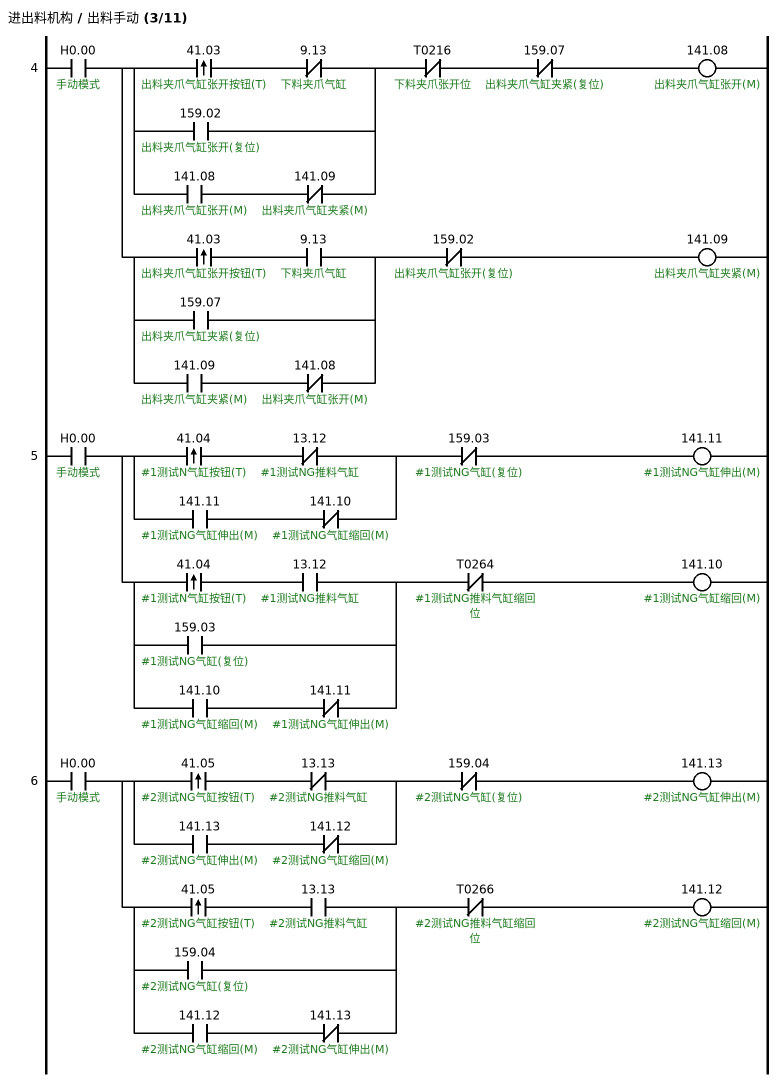
; [picture p96: 进出料机构 / 出料手动, rungs 4-6]
; rung 4
LD H0.00  ; 手动模式
OUT TR0
@LD 41.03  ; 出料夹爪气缸张开按钮(T)
ANDNOT 9.13  ; 下料夹爪气缸
OR 159.02  ; 出料夹爪气缸张开(复位)
LD 141.08  ; 出料夹爪气缸张开(M)
ANDNOT 141.09  ; 出料夹爪气缸夹紧(M)
ORLD
ANDLD
ANDNOT T0216  ; 下料夹爪张开位
ANDNOT 159.07  ; 出料夹爪气缸夹紧(复位)
OUT 141.08  ; 出料夹爪气缸张开(M)
LD TR0
@LD 41.03  ; 出料夹爪气缸张开按钮(T)
AND 9.13  ; 下料夹爪气缸
OR 159.07  ; 出料夹爪气缸夹紧(复位)
LD 141.09  ; 出料夹爪气缸夹紧(M)
ANDNOT 141.08  ; 出料夹爪气缸张开(M)
ORLD
ANDLD
ANDNOT 159.02  ; 出料夹爪气缸张开(复位)
OUT 141.09  ; 出料夹爪气缸夹紧(M)
; rung 5
LD H0.00  ; 手动模式
OUT TR0
@LD 41.04  ; #1测试N气缸按钮(T)
ANDNOT 13.12  ; #1测试NG推料气缸
LD 141.11  ; #1测试NG气缸伸出(M)
ANDNOT 141.10  ; #1测试NG气缸缩回(M)
ORLD
ANDLD
ANDNOT 159.03  ; #1测试NG气缸(复位)
OUT 141.11  ; #1测试NG气缸伸出(M)
LD TR0
@LD 41.04  ; #1测试N气缸按钮(T)
AND 13.12  ; #1测试NG推料气缸
OR 159.03  ; #1测试NG气缸(复位)
LD 141.10  ; #1测试NG气缸缩回(M)
ANDNOT 141.11  ; #1测试NG气缸伸出(M)
ORLD
ANDLD
ANDNOT T0264  ; #1测试NG推料气缸缩回位
OUT 141.10  ; #1测试NG气缸缩回(M)
; rung 6
LD H0.00  ; 手动模式
OUT TR0
@LD 41.05  ; #2测试NG气缸按钮(T)
ANDNOT 13.13  ; #2测试NG推料气缸
LD 141.13  ; #2测试NG气缸伸出(M)
ANDNOT 141.12  ; #2测试NG气缸缩回(M)
ORLD
ANDLD
ANDNOT 159.04  ; #2测试NG气缸(复位)
OUT 141.13  ; #2测试NG气缸伸出(M)
LD TR0
@LD 41.05  ; #2测试NG气缸按钮(T)
AND 13.13  ; #2测试NG推料气缸
OR 159.04  ; #2测试NG气缸(复位)
LD 141.12  ; #2测试NG气缸缩回(M)
ANDNOT 141.13  ; #2测试NG气缸伸出(M)
ORLD
ANDLD
ANDNOT T0266  ; #2测试NG推料气缸缩回位
OUT 141.12  ; #2测试NG气缸缩回(M)

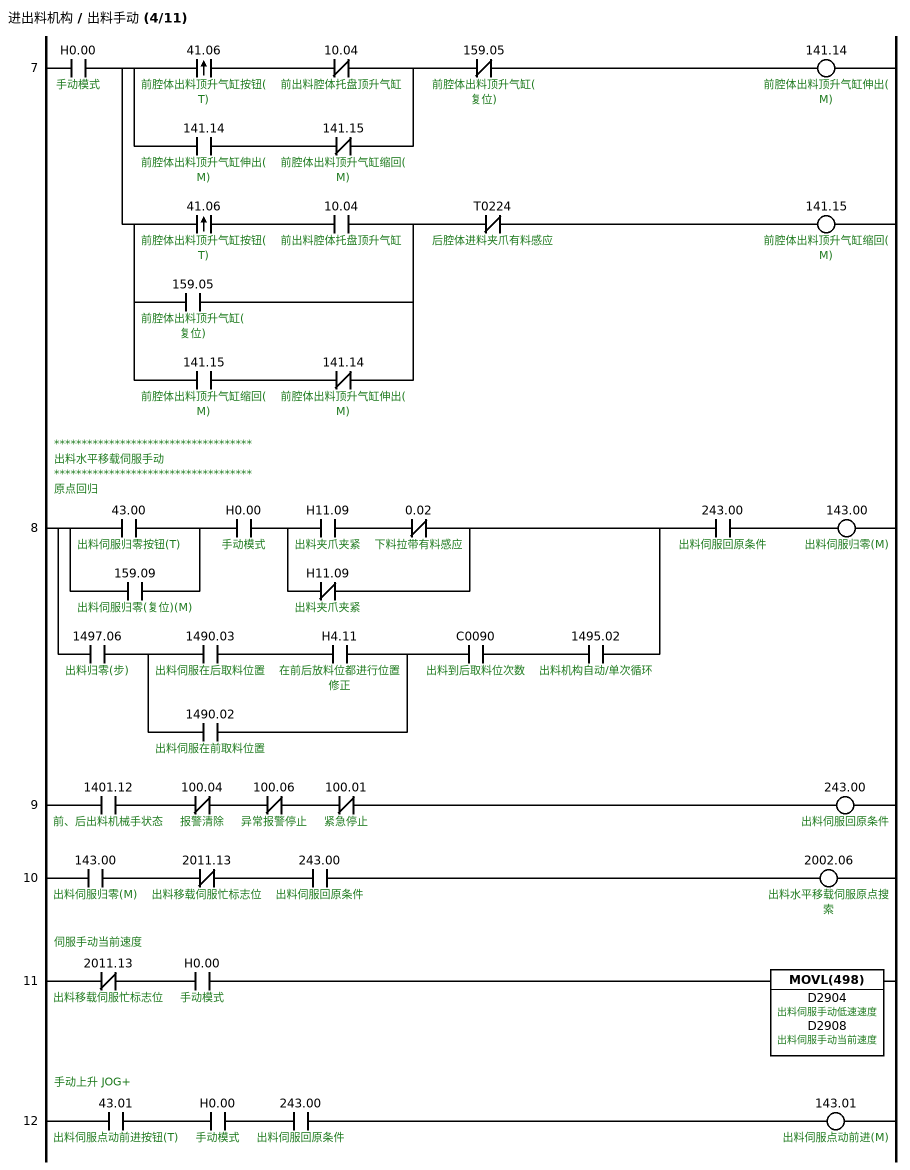
; rung 7
LD H0.00  ; 手动模式
OUT TR0
@LD 41.06  ; 前腔体出料顶升气缸按钮(T)
ANDNOT 10.04  ; 前出料腔体托盘顶升气缸
LD 141.14  ; 前腔体出料顶升气缸伸出(M)
ANDNOT 141.15  ; 前腔体出料顶升气缸缩回(M)
ORLD
ANDLD
ANDNOT 159.05  ; 前腔体出料顶升气缸(复位)
OUT 141.14  ; 前腔体出料顶升气缸伸出(M)
LD TR0
@LD 41.06  ; 前腔体出料顶升气缸按钮(T)
AND 10.04  ; 前出料腔体托盘顶升气缸
OR 159.05  ; 前腔体出料顶升气缸(复位)
LD 141.15  ; 前腔体出料顶升气缸缩回(M)
ANDNOT 141.14  ; 前腔体出料顶升气缸伸出(M)
ORLD
ANDLD
ANDNOT T0224  ; 后腔体进料夹爪有料感应
OUT 141.15  ; 前腔体出料顶升气缸缩回(M)
; rung 8: ************************************ / 出料水平移载伺服手动 / ************************************ / 原点回归
LD 43.00  ; 出料伺服归零按钮(T)
OR 159.09  ; 出料伺服归零(复位)(M)
AND H0.00  ; 手动模式
LD H11.09  ; 出料夹爪夹紧
ANDNOT 0.02  ; 下料拉带有料感应
ORNOT H11.09  ; 出料夹爪夹紧
ANDLD
LD 1497.06  ; 出料归零(步)
LD 1490.03  ; 出料伺服在后取料位置
AND H4.11  ; 在前后放料位都进行位置修正
OR 1490.02  ; 出料伺服在前取料位置
ANDLD
AND C0090  ; 出料到后取料位次数
AND 1495.02  ; 出料机构自动/单次循环
ORLD
AND 243.00  ; 出料伺服回原条件
OUT 143.00  ; 出料伺服归零(M)
; rung 9
LD 1401.12  ; 前、后出料机械手状态
ANDNOT 100.04  ; 报警清除
ANDNOT 100.06  ; 异常报警停止
ANDNOT 100.01  ; 紧急停止
OUT 243.00  ; 出料伺服回原条件
; rung 10
LD 143.00  ; 出料伺服归零(M)
ANDNOT 2011.13  ; 出料移载伺服忙标志位
AND 243.00  ; 出料伺服回原条件
OUT 2002.06  ; 出料水平移载伺服原点搜索
; rung 11: 伺服手动当前速度
LDNOT 2011.13  ; 出料移载伺服忙标志位
AND H0.00  ; 手动模式
MOVL(498) D2904 D2908  ; 出料伺服手动低速速度, 出料伺服手动当前速度
; rung 12: 手动上升 JOG+
LD 43.01  ; 出料伺服点动前进按钮(T)
AND H0.00  ; 手动模式
AND 243.00  ; 出料伺服回原条件
OUT 143.01  ; 出料伺服点动前进(M)

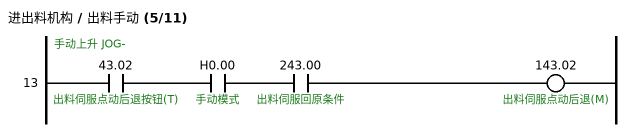
; rung 13: 手动上升 JOG-
LD 43.02  ; 出料伺服点动后退按钮(T)
AND H0.00  ; 手动模式
AND 243.00  ; 出料伺服回原条件
OUT 143.02  ; 出料伺服点动后退(M)

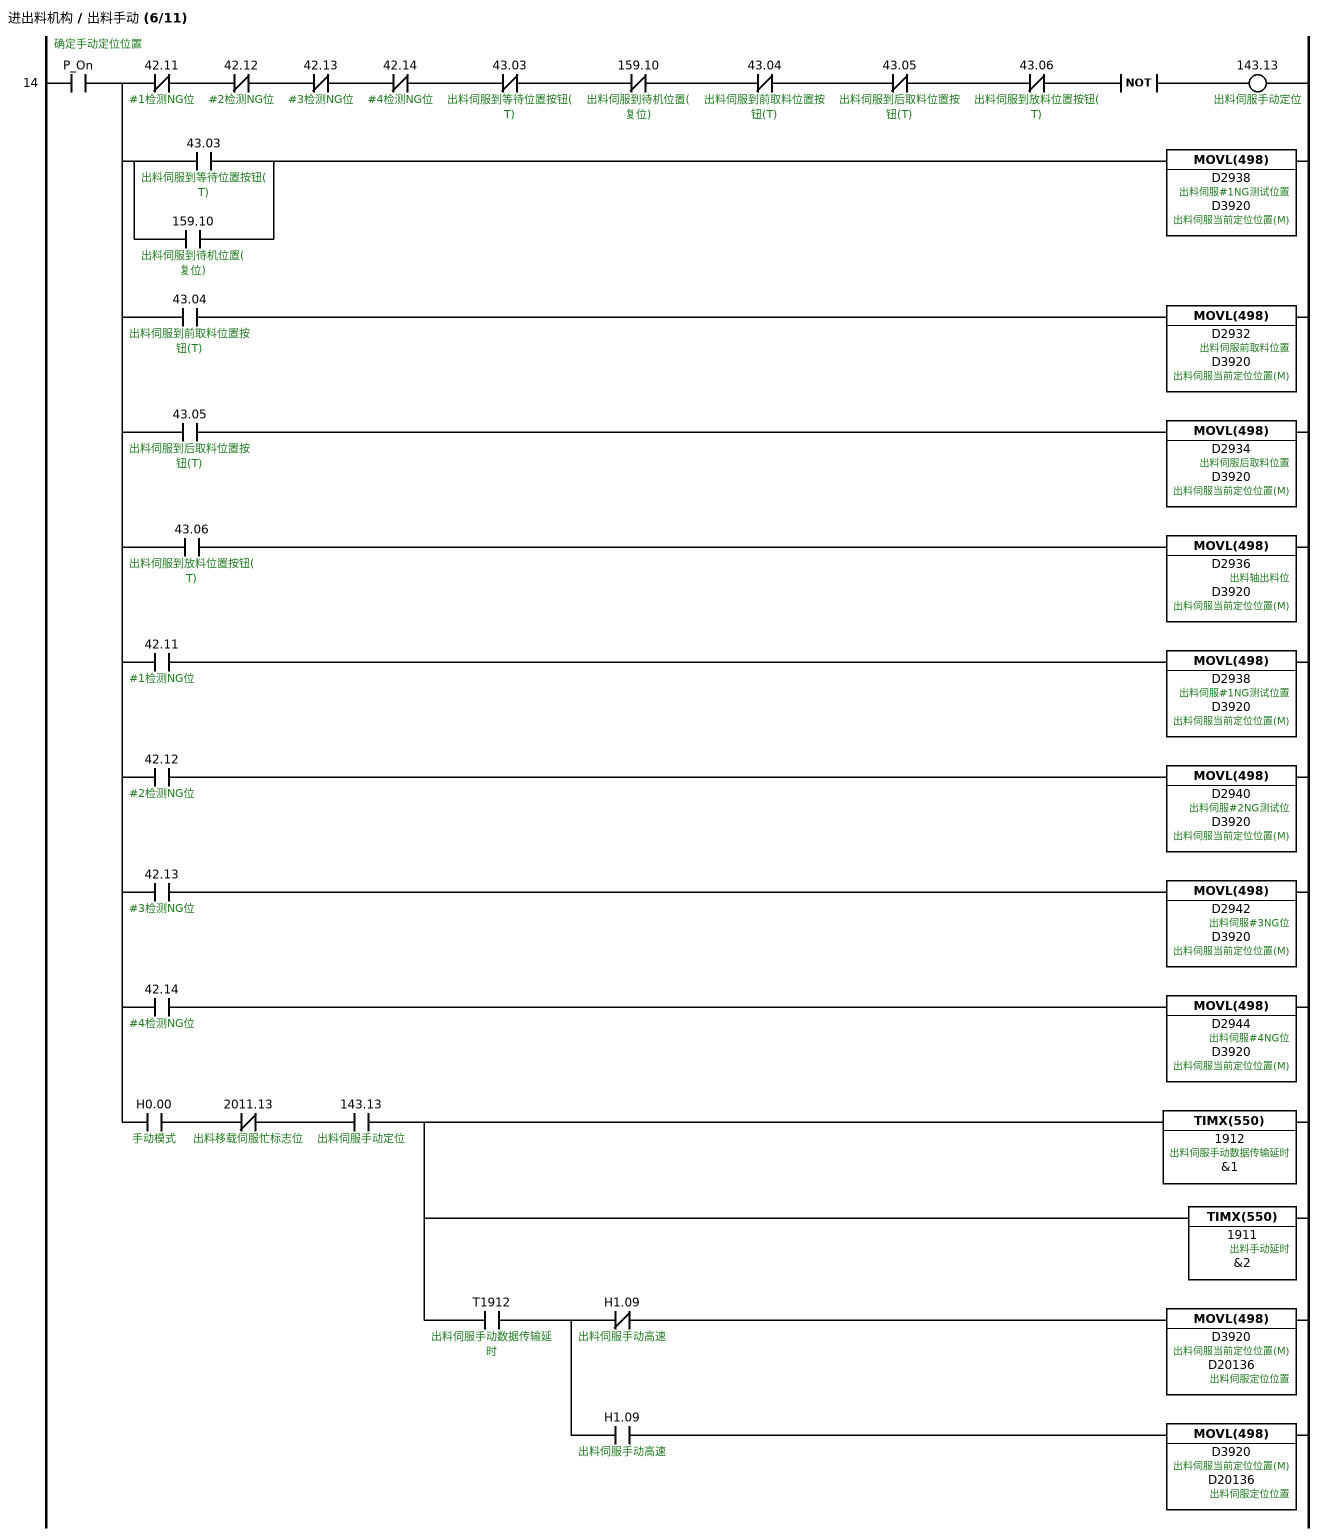
; rung 14: 确定手动定位位置
LD P_On
OUT TR0
ANDNOT 42.11  ; #1检测NG位
ANDNOT 42.12  ; #2检测NG位
ANDNOT 42.13  ; #3检测NG位
ANDNOT 42.14  ; #4检测NG位
ANDNOT 43.03  ; 出料伺服到等待位置按钮(T)
ANDNOT 159.10  ; 出料伺服到待机位置(复位)
ANDNOT 43.04  ; 出料伺服到前取料位置按钮(T)
ANDNOT 43.05  ; 出料伺服到后取料位置按钮(T)
ANDNOT 43.06  ; 出料伺服到放料位置按钮(T)
NOT(520)
OUT 143.13  ; 出料伺服手动定位
LD TR0
LD 43.03  ; 出料伺服到等待位置按钮(T)
OR 159.10  ; 出料伺服到待机位置(复位)
ANDLD
MOVL(498) D2938 D3920  ; 出料伺服#1NG测试位置, 出料伺服当前定位位置(M)
LD TR0
AND 43.04  ; 出料伺服到前取料位置按钮(T)
MOVL(498) D2932 D3920  ; 出料伺服前取料位置, 出料伺服当前定位位置(M)
LD TR0
AND 43.05  ; 出料伺服到后取料位置按钮(T)
MOVL(498) D2934 D3920  ; 出料伺服后取料位置, 出料伺服当前定位位置(M)
LD TR0
AND 43.06  ; 出料伺服到放料位置按钮(T)
MOVL(498) D2936 D3920  ; 出料轴出料位, 出料伺服当前定位位置(M)
LD TR0
AND 42.11  ; #1检测NG位
MOVL(498) D2938 D3920  ; 出料伺服#1NG测试位置, 出料伺服当前定位位置(M)
LD TR0
AND 42.12  ; #2检测NG位
MOVL(498) D2940 D3920  ; 出料伺服#2NG测试位, 出料伺服当前定位位置(M)
LD TR0
AND 42.13  ; #3检测NG位
MOVL(498) D2942 D3920  ; 出料伺服#3NG位, 出料伺服当前定位位置(M)
LD TR0
AND 42.14  ; #4检测NG位
MOVL(498) D2944 D3920  ; 出料伺服#4NG位, 出料伺服当前定位位置(M)
LD TR0
AND H0.00  ; 手动模式
ANDNOT 2011.13  ; 出料移载伺服忙标志位
AND 143.13  ; 出料伺服手动定位
TIMX(550) 1912 &1  ; 出料伺服手动数据传输延时
TIMX(550) 1911 &2  ; 出料手动延时
AND T1912  ; 出料伺服手动数据传输延时
OUT TR0
ANDNOT H1.09  ; 出料伺服手动高速
MOVL(498) D3920 D20136  ; 出料伺服当前定位位置(M), 出料伺服定位位置
LD TR0
AND H1.09  ; 出料伺服手动高速
MOVL(498) D3920 D20136  ; 出料伺服当前定位位置(M), 出料伺服定位位置

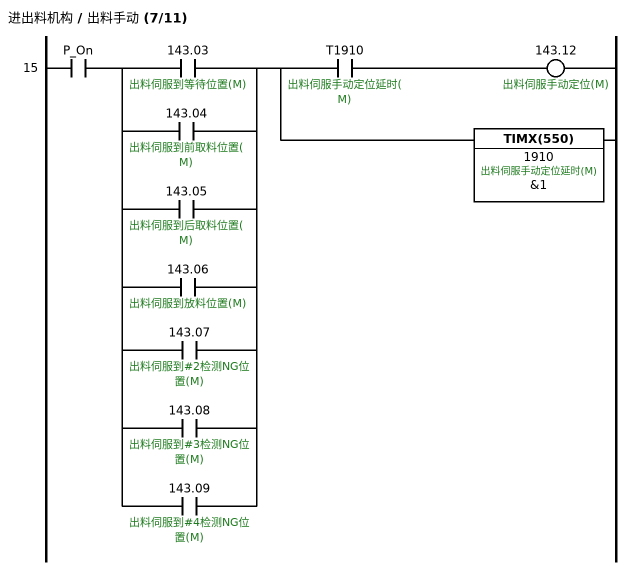
; rung 15
LD P_On
LD 143.03  ; 出料伺服到等待位置(M)
OR 143.04  ; 出料伺服到前取料位置(M)
OR 143.05  ; 出料伺服到后取料位置(M)
OR 143.06  ; 出料伺服到放料位置(M)
OR 143.07  ; 出料伺服到#2检测NG位置(M)
OR 143.08  ; 出料伺服到#3检测NG位置(M)
OR 143.09  ; 出料伺服到#4检测NG位置(M)
ANDLD
OUT TR0
AND T1910  ; 出料伺服手动定位延时(M)
OUT 143.12  ; 出料伺服手动定位(M)
LD TR0
TIMX(550) 1910 &1  ; 出料伺服手动定位延时(M)

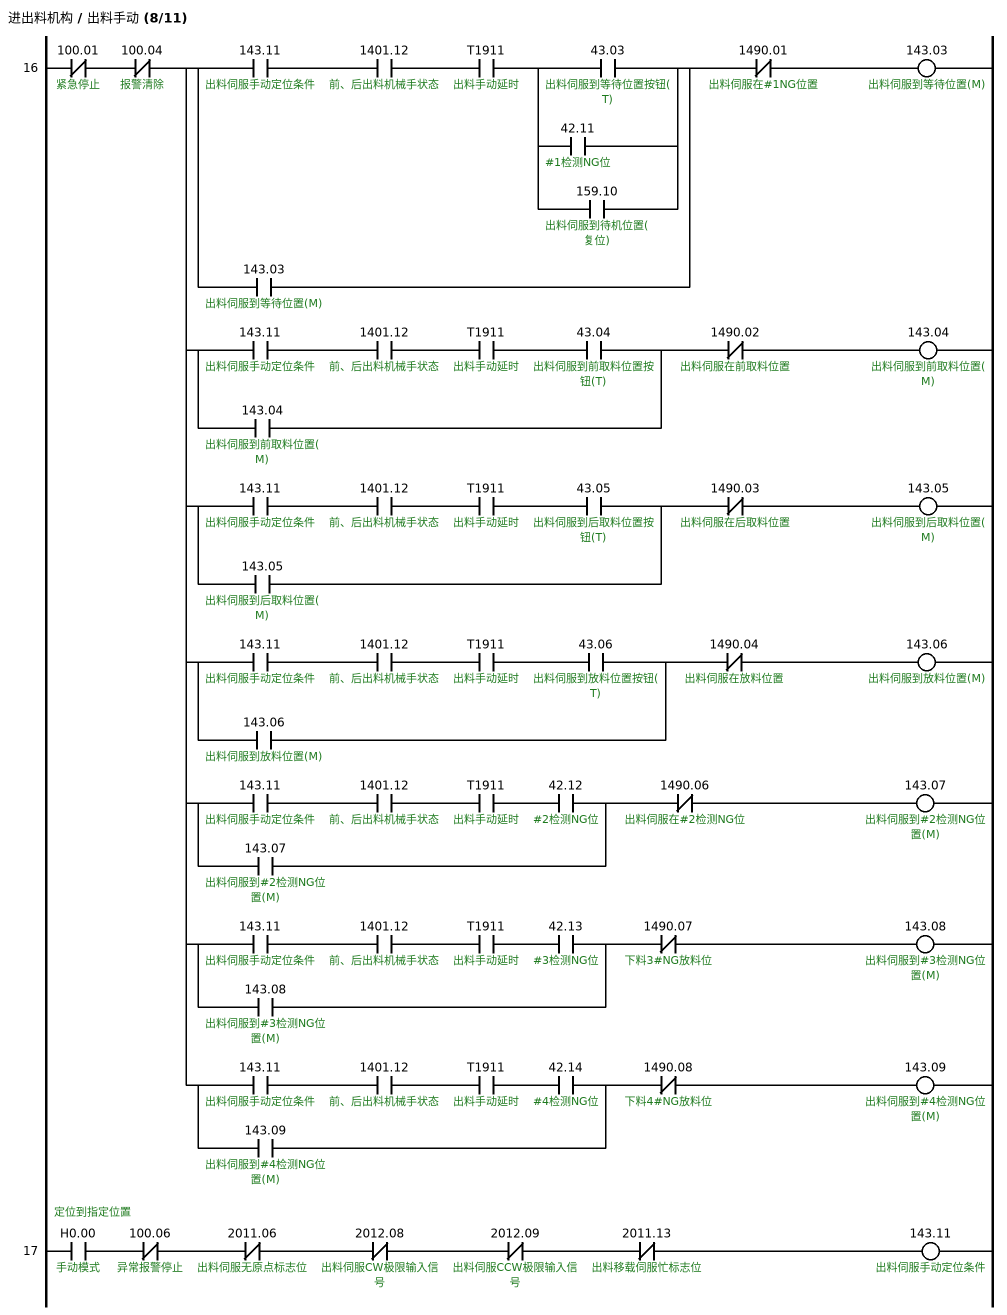
; rung 16
LDNOT 100.01  ; 紧急停止
ANDNOT 100.04  ; 报警清除
OUT TR0
LD 143.11  ; 出料伺服手动定位条件
AND 1401.12  ; 前、后出料机械手状态
AND T1911  ; 出料手动延时
LD 43.03  ; 出料伺服到等待位置按钮(T)
OR 42.11  ; #1检测NG位
OR 159.10  ; 出料伺服到待机位置(复位)
ANDLD
OR 143.03  ; 出料伺服到等待位置(M)
ANDLD
ANDNOT 1490.01  ; 出料伺服在#1NG位置
OUT 143.03  ; 出料伺服到等待位置(M)
LD TR0
LD 143.11  ; 出料伺服手动定位条件
AND 1401.12  ; 前、后出料机械手状态
AND T1911  ; 出料手动延时
AND 43.04  ; 出料伺服到前取料位置按钮(T)
OR 143.04  ; 出料伺服到前取料位置(M)
ANDLD
ANDNOT 1490.02  ; 出料伺服在前取料位置
OUT 143.04  ; 出料伺服到前取料位置(M)
LD TR0
LD 143.11  ; 出料伺服手动定位条件
AND 1401.12  ; 前、后出料机械手状态
AND T1911  ; 出料手动延时
AND 43.05  ; 出料伺服到后取料位置按钮(T)
OR 143.05  ; 出料伺服到后取料位置(M)
ANDLD
ANDNOT 1490.03  ; 出料伺服在后取料位置
OUT 143.05  ; 出料伺服到后取料位置(M)
LD TR0
LD 143.11  ; 出料伺服手动定位条件
AND 1401.12  ; 前、后出料机械手状态
AND T1911  ; 出料手动延时
AND 43.06  ; 出料伺服到放料位置按钮(T)
OR 143.06  ; 出料伺服到放料位置(M)
ANDLD
ANDNOT 1490.04  ; 出料伺服在放料位置
OUT 143.06  ; 出料伺服到放料位置(M)
LD TR0
LD 143.11  ; 出料伺服手动定位条件
AND 1401.12  ; 前、后出料机械手状态
AND T1911  ; 出料手动延时
AND 42.12  ; #2检测NG位
OR 143.07  ; 出料伺服到#2检测NG位置(M)
ANDLD
ANDNOT 1490.06  ; 出料伺服在#2检测NG位
OUT 143.07  ; 出料伺服到#2检测NG位置(M)
LD TR0
LD 143.11  ; 出料伺服手动定位条件
AND 1401.12  ; 前、后出料机械手状态
AND T1911  ; 出料手动延时
AND 42.13  ; #3检测NG位
OR 143.08  ; 出料伺服到#3检测NG位置(M)
ANDLD
ANDNOT 1490.07  ; 下料3#NG放料位
OUT 143.08  ; 出料伺服到#3检测NG位置(M)
LD TR0
LD 143.11  ; 出料伺服手动定位条件
AND 1401.12  ; 前、后出料机械手状态
AND T1911  ; 出料手动延时
AND 42.14  ; #4检测NG位
OR 143.09  ; 出料伺服到#4检测NG位置(M)
ANDLD
ANDNOT 1490.08  ; 下料4#NG放料位
OUT 143.09  ; 出料伺服到#4检测NG位置(M)
; rung 17: 定位到指定位置
LD H0.00  ; 手动模式
ANDNOT 100.06  ; 异常报警停止
ANDNOT 2011.06  ; 出料伺服无原点标志位
ANDNOT 2012.08  ; 出料伺服CW极限输入信号
ANDNOT 2012.09  ; 出料伺服CCW极限输入信号
ANDNOT 2011.13  ; 出料移载伺服忙标志位
OUT 143.11  ; 出料伺服手动定位条件

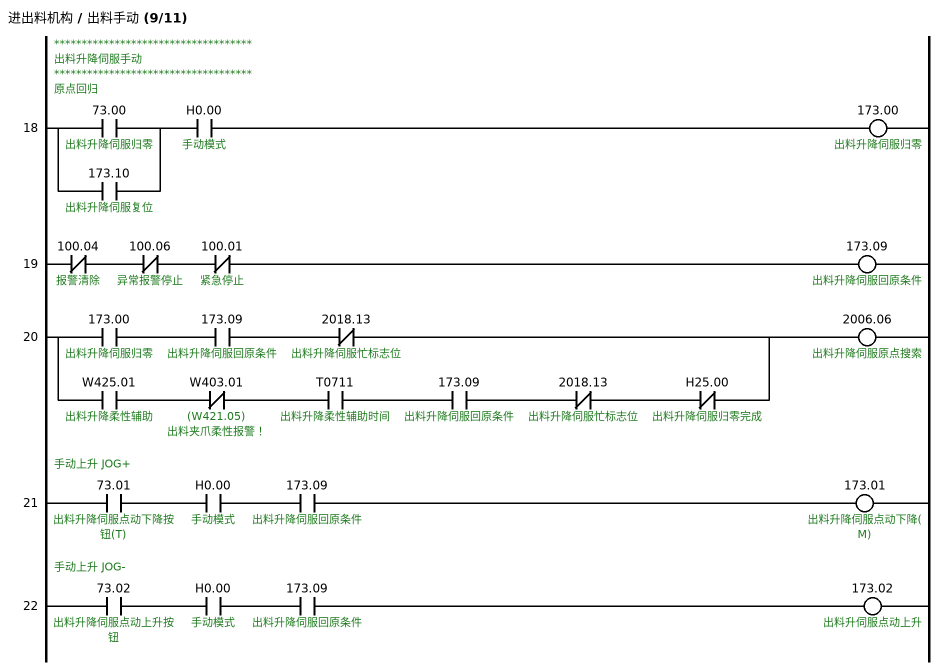
; rung 18: ************************************ / 出料升降伺服手动 / ************************************ / 原点回归
LD 73.00  ; 出料升降伺服归零
OR 173.10  ; 出料升降伺服复位
AND H0.00  ; 手动模式
OUT 173.00  ; 出料升降伺服归零
; rung 19
LDNOT 100.04  ; 报警清除
ANDNOT 100.06  ; 异常报警停止
ANDNOT 100.01  ; 紧急停止
OUT 173.09  ; 出料升降伺服回原条件
; rung 20
LD 173.00  ; 出料升降伺服归零
AND 173.09  ; 出料升降伺服回原条件
ANDNOT 2018.13  ; 出料升降伺服忙标志位
LD W425.01  ; 出料升降柔性辅助
ANDNOT W403.01  ; (W421.05) 出料夹爪柔性报警！
AND T0711  ; 出料升降柔性辅助时间
AND 173.09  ; 出料升降伺服回原条件
ANDNOT 2018.13  ; 出料升降伺服忙标志位
ANDNOT H25.00  ; 出料升降伺服归零完成
ORLD
OUT 2006.06  ; 出料升降伺服原点搜索
; rung 21: 手动上升 JOG+
LD 73.01  ; 出料升降伺服点动下降按钮(T)
AND H0.00  ; 手动模式
AND 173.09  ; 出料升降伺服回原条件
OUT 173.01  ; 出料升降伺服点动下降(M)
; rung 22: 手动上升 JOG-
LD 73.02  ; 出料升降伺服点动上升按钮
AND H0.00  ; 手动模式
AND 173.09  ; 出料升降伺服回原条件
OUT 173.02  ; 出料升伺服点动上升

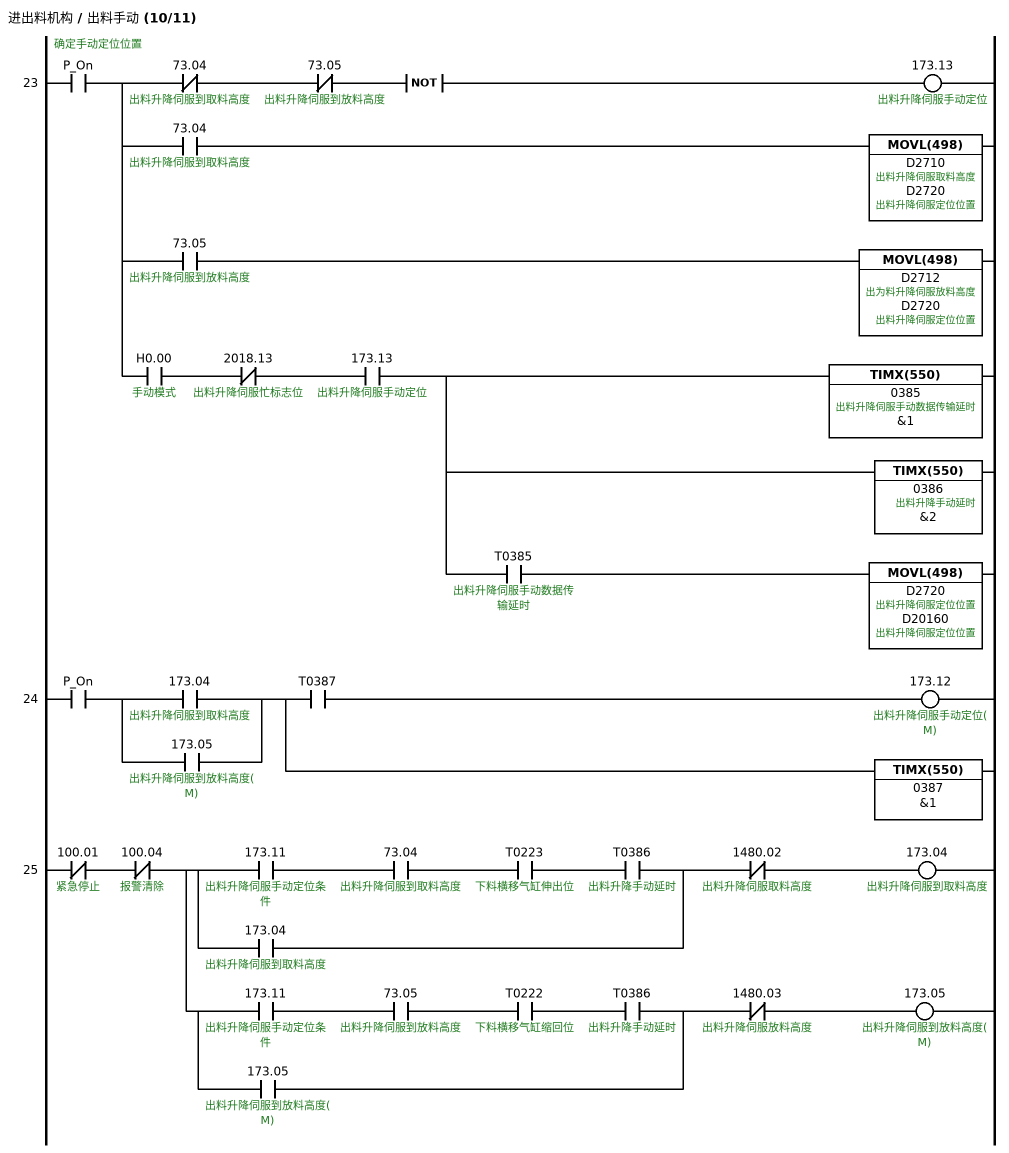
; rung 23: 确定手动定位位置
LD P_On
OUT TR0
ANDNOT 73.04  ; 出料升降伺服到取料高度
ANDNOT 73.05  ; 出料升降伺服到放料高度
NOT(520)
OUT 173.13  ; 出料升降伺服手动定位
LD TR0
AND 73.04  ; 出料升降伺服到取料高度
MOVL(498) D2710 D2720  ; 出料升降伺服取料高度, 出料升降伺服定位位置
LD TR0
AND 73.05  ; 出料升降伺服到放料高度
MOVL(498) D2712 D2720  ; 出为料升降伺服放料高度, 出料升降伺服定位位置
LD TR0
AND H0.00  ; 手动模式
ANDNOT 2018.13  ; 出料升降伺服忙标志位
AND 173.13  ; 出料升降伺服手动定位
TIMX(550) 0385 &1  ; 出料升降伺服手动数据传输延时
TIMX(550) 0386 &2  ; 出料升降手动延时
AND T0385  ; 出料升降伺服手动数据传输延时
MOVL(498) D2720 D20160  ; 出料升降伺服定位位置
; rung 24
LD P_On
LD 173.04  ; 出料升降伺服到取料高度
OR 173.05  ; 出料升降伺服到放料高度(M)
ANDLD
OUT TR0
AND T0387
OUT 173.12  ; 出料升降伺服手动定位(M)
LD TR0
TIMX(550) 0387 &1
; rung 25
LDNOT 100.01  ; 紧急停止
ANDNOT 100.04  ; 报警清除
OUT TR0
LD 173.11  ; 出料升降伺服手动定位条件
AND 73.04  ; 出料升降伺服到取料高度
AND T0223  ; 下料横移气缸伸出位
AND T0386  ; 出料升降手动延时
OR 173.04  ; 出料升降伺服到取料高度
ANDLD
ANDNOT 1480.02  ; 出料升降伺服取料高度
OUT 173.04  ; 出料升降伺服到取料高度
LD TR0
LD 173.11  ; 出料升降伺服手动定位条件
AND 73.05  ; 出料升降伺服到放料高度
AND T0222  ; 下料横移气缸缩回位
AND T0386  ; 出料升降手动延时
OR 173.05  ; 出料升降伺服到放料高度(M)
ANDLD
ANDNOT 1480.03  ; 出料升降伺服放料高度
OUT 173.05  ; 出料升降伺服到放料高度(M)

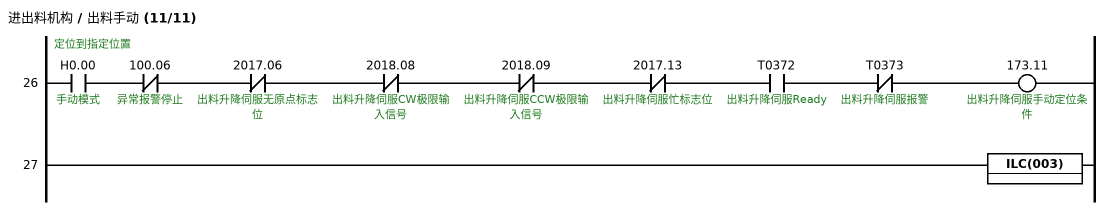
; rung 26: 定位到指定位置
LD H0.00  ; 手动模式
ANDNOT 100.06  ; 异常报警停止
ANDNOT 2017.06  ; 出料升降伺服无原点标志位
ANDNOT 2018.08  ; 出料升降伺服CW极限输入信号
ANDNOT 2018.09  ; 出料升降伺服CCW极限输入信号
ANDNOT 2017.13  ; 出料升降伺服忙标志位
AND T0372  ; 出料升降伺服Ready
ANDNOT T0373  ; 出料升降伺服报警
OUT 173.11  ; 出料升降伺服手动定位条件
; rung 27
ILC(003)

### Section 出料自动

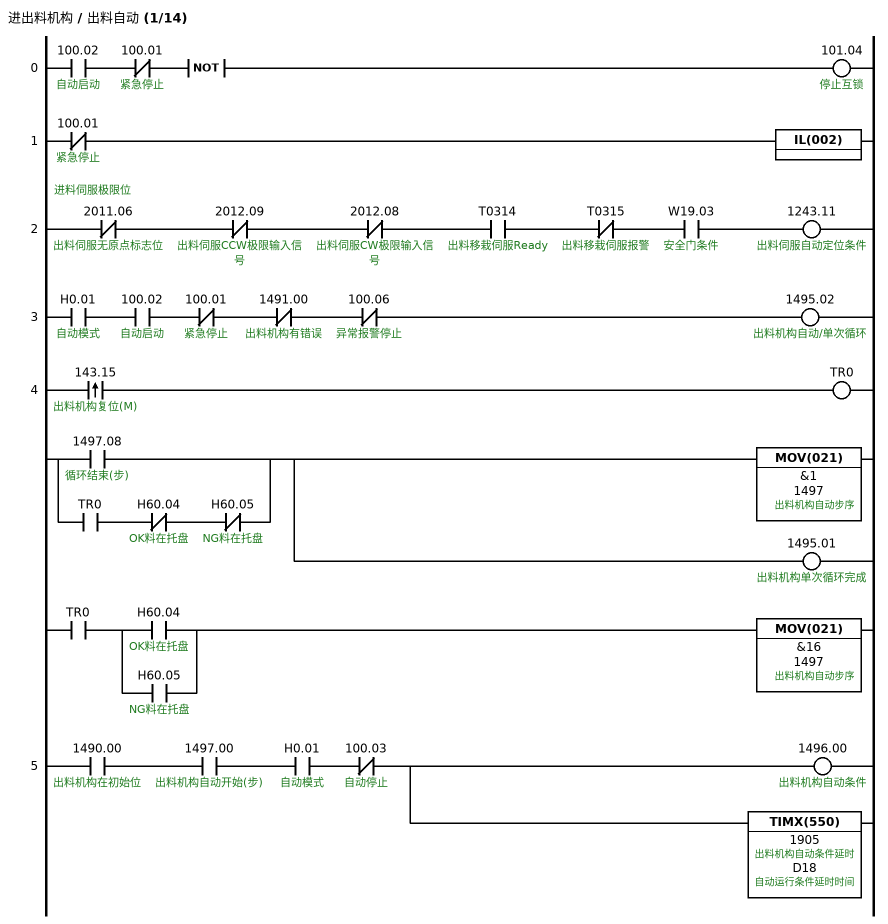
; rung 0
LD 100.02  ; 自动启动
ANDNOT 100.01  ; 紧急停止
NOT(520)
OUT 101.04  ; 停止互锁
; rung 1
LDNOT 100.01  ; 紧急停止
IL(002)
; rung 2: 进料伺服极限位
LDNOT 2011.06  ; 出料伺服无原点标志位
ANDNOT 2012.09  ; 出料伺服CCW极限输入信号
ANDNOT 2012.08  ; 出料伺服CW极限输入信号
AND T0314  ; 出料移栽伺服Ready
ANDNOT T0315  ; 出料移栽伺服报警
AND W19.03  ; 安全门条件
OUT 1243.11  ; 出料伺服自动定位条件
; rung 3
LD H0.01  ; 自动模式
AND 100.02  ; 自动启动
ANDNOT 100.01  ; 紧急停止
ANDNOT 1491.00  ; 出料机构有错误
ANDNOT 100.06  ; 异常报警停止
OUT 1495.02  ; 出料机构自动/单次循环
; rung 4
LD 1497.08  ; 循环结束(步)
@LD 143.15  ; 出料机构复位(M)
OUT TR0
ANDNOT H60.04  ; OK料在托盘
ANDNOT H60.05  ; NG料在托盘
ORLD
MOV(021) &1 1497  ; 出料机构自动步序
OUT 1495.01  ; 出料机构单次循环完成
LD TR0
LD H60.04  ; OK料在托盘
OR H60.05  ; NG料在托盘
ANDLD
MOV(021) &16 1497  ; 出料机构自动步序
; rung 5
LD 1490.00  ; 出料机构在初始位
AND 1497.00  ; 出料机构自动开始(步)
AND H0.01  ; 自动模式
ANDNOT 100.03  ; 自动停止
OUT 1496.00  ; 出料机构自动条件
TIMX(550) 1905 D18  ; 自动运行条件延时时间, 出料机构自动条件延时

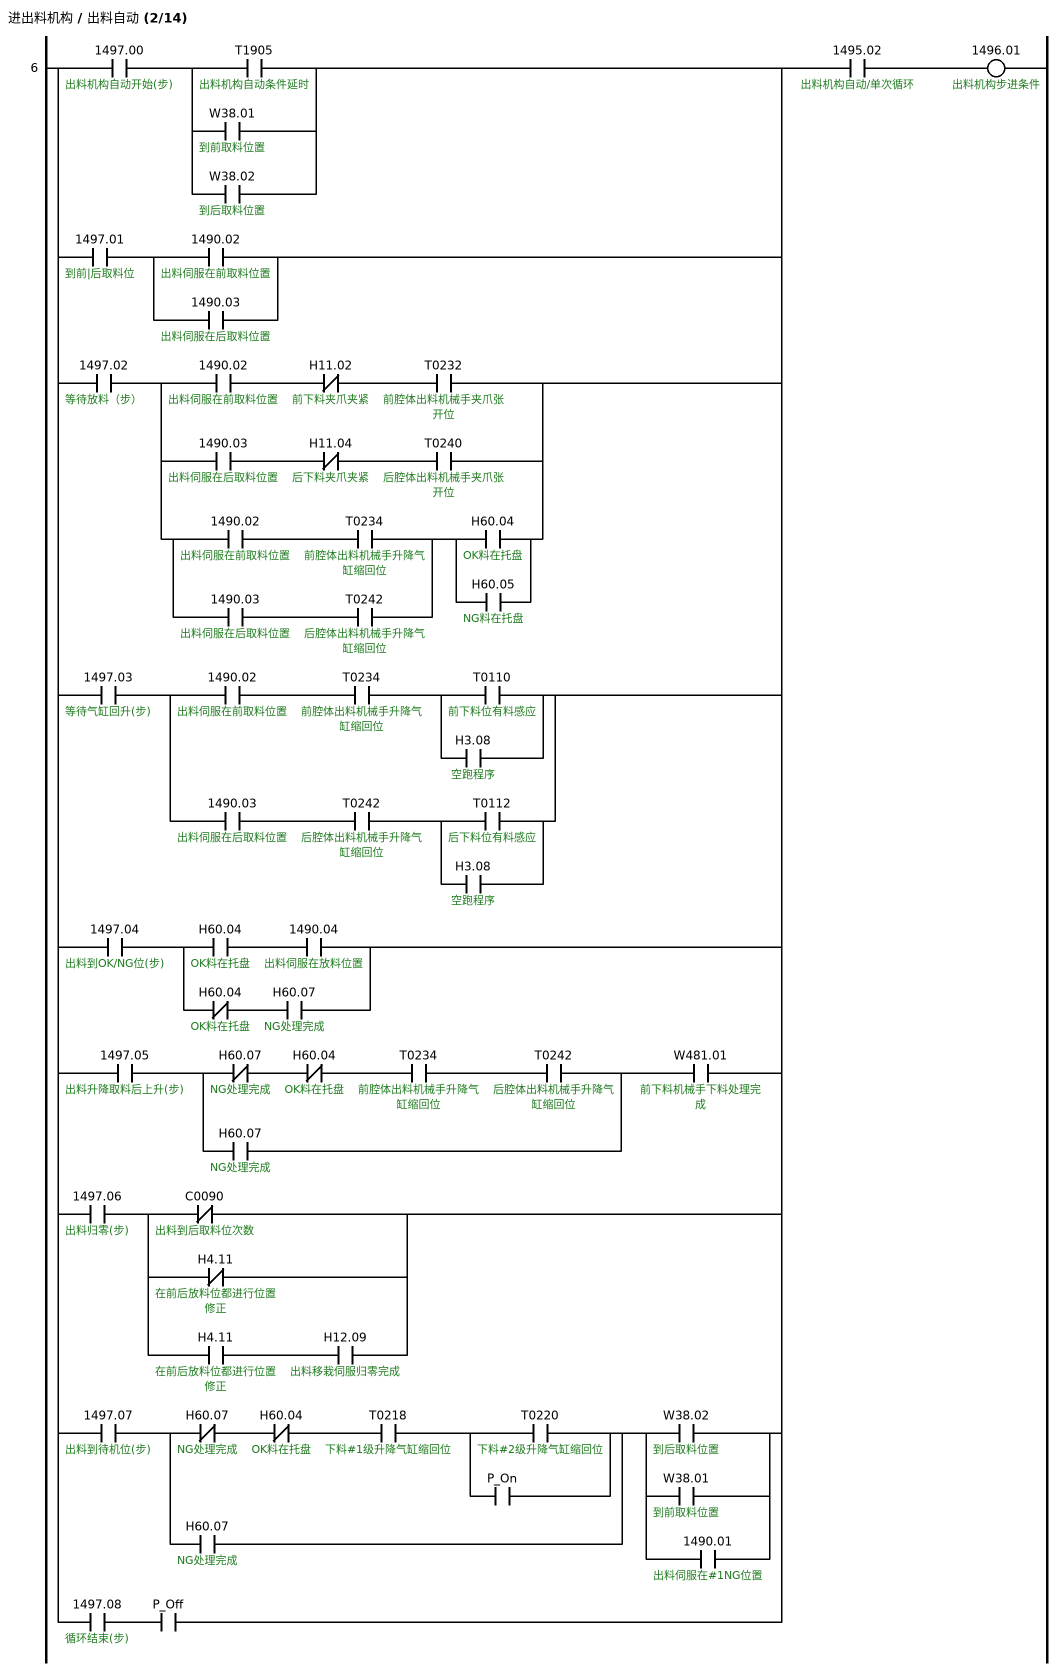
; rung 6
LD 1497.00  ; 出料机构自动开始(步)
LD T1905  ; 出料机构自动条件延时
OR W38.01  ; 到前取料位置
OR W38.02  ; 到后取料位置
ANDLD
LD 1497.01  ; 到前|后取料位
LD 1490.02  ; 出料伺服在前取料位置
OR 1490.03  ; 出料伺服在后取料位置
ANDLD
ORLD
LD 1497.02  ; 等待放料（步）
LD 1490.02  ; 出料伺服在前取料位置
ANDNOT H11.02  ; 前下料夹爪夹紧
AND T0232  ; 前腔体出料机械手夹爪张开位
LD 1490.03  ; 出料伺服在后取料位置
ANDNOT H11.04  ; 后下料夹爪夹紧
AND T0240  ; 后腔体出料机械手夹爪张开位
ORLD
LD 1490.02  ; 出料伺服在前取料位置
AND T0234  ; 前腔体出料机械手升降气缸缩回位
LD 1490.03  ; 出料伺服在后取料位置
AND T0242  ; 后腔体出料机械手升降气缸缩回位
ORLD
LD H60.04  ; OK料在托盘
OR H60.05  ; NG料在托盘
ANDLD
ORLD
ANDLD
ORLD
LD 1497.03  ; 等待气缸回升(步)
LD 1490.02  ; 出料伺服在前取料位置
AND T0234  ; 前腔体出料机械手升降气缸缩回位
LD T0110  ; 前下料位有料感应
OR H3.08  ; 空跑程序
ANDLD
LD 1490.03  ; 出料伺服在后取料位置
AND T0242  ; 后腔体出料机械手升降气缸缩回位
LD T0112  ; 后下料位有料感应
OR H3.08  ; 空跑程序
ANDLD
ORLD
ANDLD
ORLD
LD 1497.04  ; 出料到OK/NG位(步)
LD H60.04  ; OK料在托盘
AND 1490.04  ; 出料伺服在放料位置
LDNOT H60.04  ; OK料在托盘
AND H60.07  ; NG处理完成
ORLD
ANDLD
ORLD
LD 1497.05  ; 出料升降取料后上升(步)
LDNOT H60.07  ; NG处理完成
ANDNOT H60.04  ; OK料在托盘
AND T0234  ; 前腔体出料机械手升降气缸缩回位
AND T0242  ; 后腔体出料机械手升降气缸缩回位
OR H60.07  ; NG处理完成
ANDLD
AND W481.01  ; 前下料机械手下料处理完成
ORLD
LD 1497.06  ; 出料归零(步)
LDNOT C0090  ; 出料到后取料位次数
ORNOT H4.11  ; 在前后放料位都进行位置修正
LD H4.11  ; 在前后放料位都进行位置修正
AND H12.09  ; 出料移栽伺服归零完成
ORLD
ANDLD
ORLD
LD 1497.07  ; 出料到待机位(步)
LDNOT H60.07  ; NG处理完成
ANDNOT H60.04  ; OK料在托盘
AND T0218  ; 下料#1级升降气缸缩回位
LD T0220  ; 下料#2级升降气缸缩回位
OR P_On
ANDLD
OR H60.07  ; NG处理完成
ANDLD
LD W38.02  ; 到后取料位置
OR W38.01  ; 到前取料位置
OR 1490.01  ; 出料伺服在#1NG位置
ANDLD
ORLD
LD 1497.08  ; 循环结束(步)
AND P_Off
ORLD
AND 1495.02  ; 出料机构自动/单次循环
OUT 1496.01  ; 出料机构步进条件

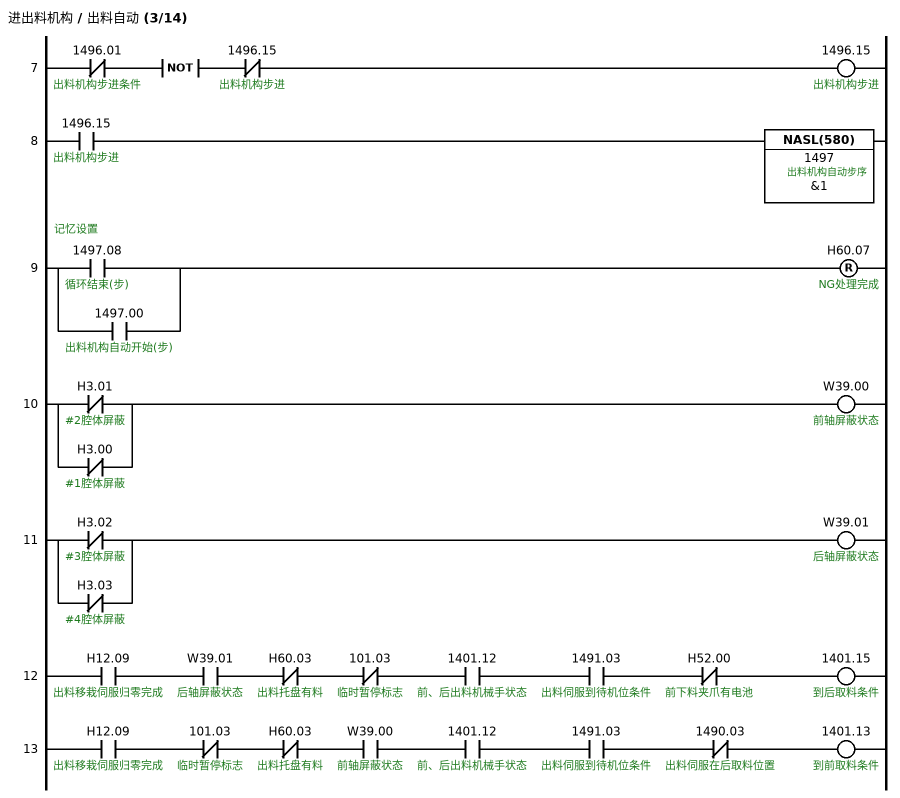
; rung 7
LDNOT 1496.01  ; 出料机构步进条件
NOT(520)
ANDNOT 1496.15  ; 出料机构步进
OUT 1496.15  ; 出料机构步进
; rung 8
LD 1496.15  ; 出料机构步进
NASL(580) 1497 &1  ; 出料机构自动步序
; rung 9: 记忆设置
LD 1497.08  ; 循环结束(步)
OR 1497.00  ; 出料机构自动开始(步)
RSET H60.07  ; NG处理完成
; rung 10
LDNOT H3.01  ; #2腔体屏蔽
ORNOT H3.00  ; #1腔体屏蔽
OUT W39.00  ; 前轴屏蔽状态
; rung 11
LDNOT H3.02  ; #3腔体屏蔽
ORNOT H3.03  ; #4腔体屏蔽
OUT W39.01  ; 后轴屏蔽状态
; rung 12
LD H12.09  ; 出料移栽伺服归零完成
AND W39.01  ; 后轴屏蔽状态
ANDNOT H60.03  ; 出料托盘有料
ANDNOT 101.03  ; 临时暂停标志
AND 1401.12  ; 前、后出料机械手状态
AND 1491.03  ; 出料伺服到待机位条件
ANDNOT H52.00  ; 前下料夹爪有电池
OUT 1401.15  ; 到后取料条件
; rung 13
LD H12.09  ; 出料移栽伺服归零完成
ANDNOT 101.03  ; 临时暂停标志
ANDNOT H60.03  ; 出料托盘有料
AND W39.00  ; 前轴屏蔽状态
AND 1401.12  ; 前、后出料机械手状态
AND 1491.03  ; 出料伺服到待机位条件
ANDNOT 1490.03  ; 出料伺服在后取料位置
OUT 1401.13  ; 到前取料条件

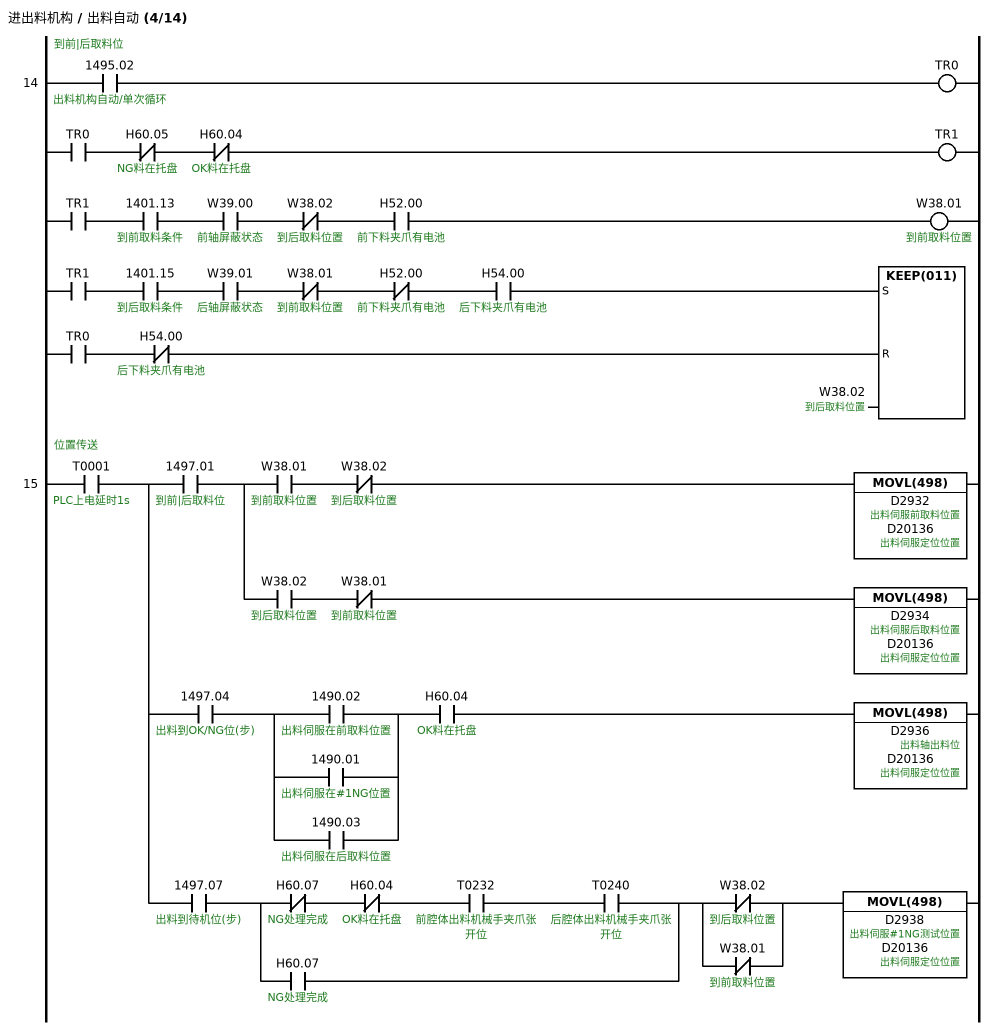
; rung 14: 到前|后取料位
LD 1495.02  ; 出料机构自动/单次循环
OUT TR0
ANDNOT H60.05  ; NG料在托盘
ANDNOT H60.04  ; OK料在托盘
OUT TR1
AND 1401.13  ; 到前取料条件
AND W39.00  ; 前轴屏蔽状态
ANDNOT W38.02  ; 到后取料位置
AND H52.00  ; 前下料夹爪有电池
OUT W38.01  ; 到前取料位置
LD TR1
AND 1401.15  ; 到后取料条件
AND W39.01  ; 后轴屏蔽状态
ANDNOT W38.01  ; 到前取料位置
ANDNOT H52.00  ; 前下料夹爪有电池
AND H54.00  ; 后下料夹爪有电池
LD TR0
ANDNOT H54.00  ; 后下料夹爪有电池
KEEP(011) W38.02  ; 到后取料位置
; rung 15: 位置传送
LD T0001  ; PLC上电延时1s
OUT TR0
AND 1497.01  ; 到前|后取料位
OUT TR1
AND W38.01  ; 到前取料位置
ANDNOT W38.02  ; 到后取料位置
MOVL(498) D2932 D20136  ; 出料伺服前取料位置, 出料伺服定位位置
LD TR1
AND W38.02  ; 到后取料位置
ANDNOT W38.01  ; 到前取料位置
MOVL(498) D2934 D20136  ; 出料伺服后取料位置, 出料伺服定位位置
LD TR0
AND 1497.04  ; 出料到OK/NG位(步)
LD 1490.02  ; 出料伺服在前取料位置
OR 1490.01  ; 出料伺服在#1NG位置
OR 1490.03  ; 出料伺服在后取料位置
ANDLD
AND H60.04  ; OK料在托盘
MOVL(498) D2936 D20136  ; 出料轴出料位, 出料伺服定位位置
LD TR0
AND 1497.07  ; 出料到待机位(步)
LDNOT H60.07  ; NG处理完成
ANDNOT H60.04  ; OK料在托盘
AND T0232  ; 前腔体出料机械手夹爪张开位
AND T0240  ; 后腔体出料机械手夹爪张开位
OR H60.07  ; NG处理完成
ANDLD
LDNOT W38.02  ; 到后取料位置
ORNOT W38.01  ; 到前取料位置
ANDLD
MOVL(498) D2938 D20136  ; 出料伺服#1NG测试位置, 出料伺服定位位置

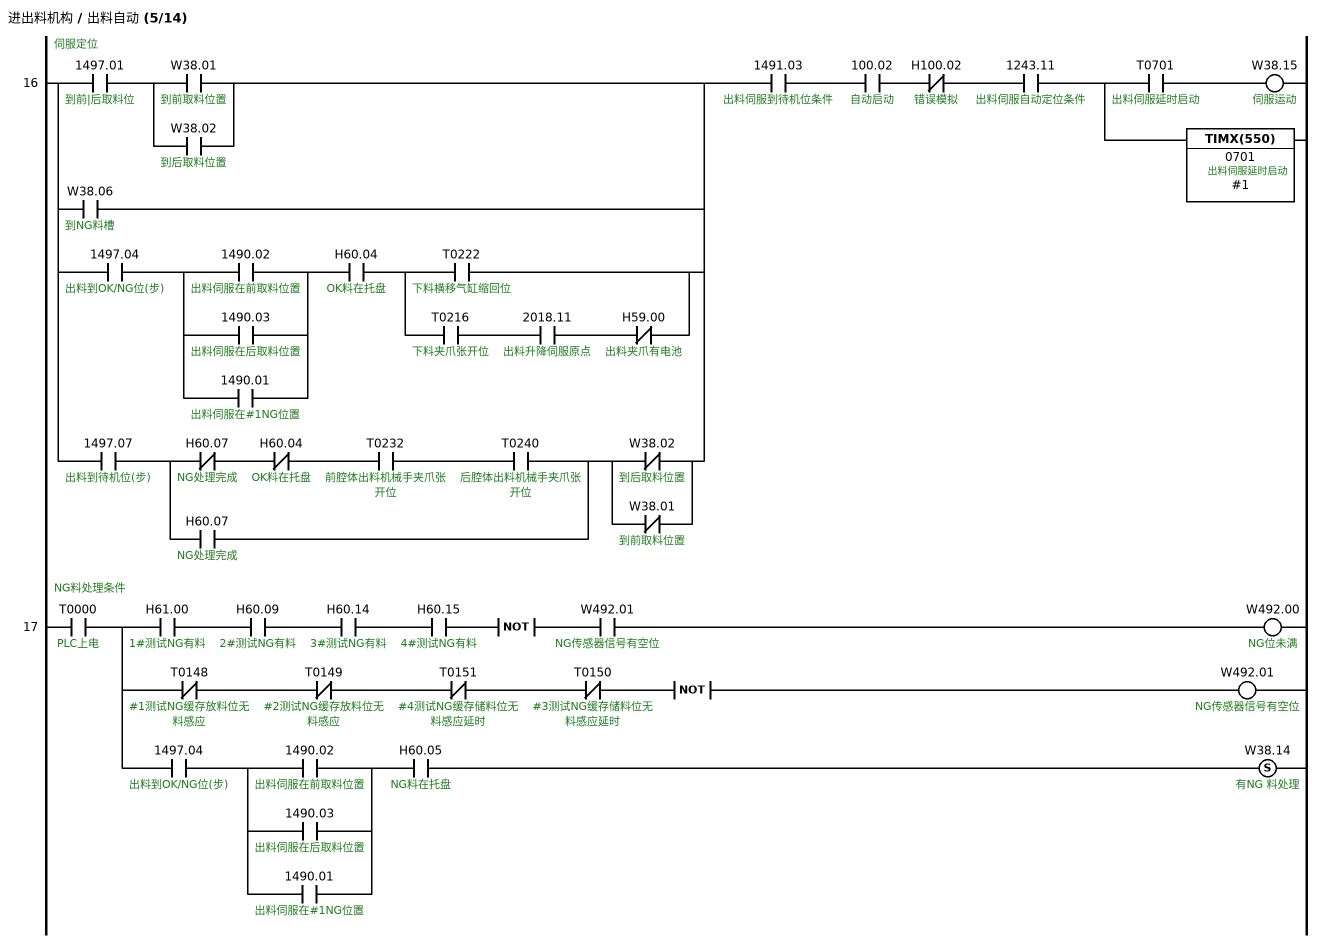
; rung 16: 伺服定位
LD 1497.01  ; 到前|后取料位
LD W38.01  ; 到前取料位置
OR W38.02  ; 到后取料位置
ANDLD
OR W38.06  ; 到NG料槽
LD 1497.04  ; 出料到OK/NG位(步)
LD 1490.02  ; 出料伺服在前取料位置
OR 1490.03  ; 出料伺服在后取料位置
OR 1490.01  ; 出料伺服在#1NG位置
ANDLD
AND H60.04  ; OK料在托盘
LD T0222  ; 下料横移气缸缩回位
LD T0216  ; 下料夹爪张开位
AND 2018.11  ; 出料升降伺服原点
ANDNOT H59.00  ; 出料夹爪有电池
ORLD
ANDLD
ORLD
LD 1497.07  ; 出料到待机位(步)
LDNOT H60.07  ; NG处理完成
ANDNOT H60.04  ; OK料在托盘
AND T0232  ; 前腔体出料机械手夹爪张开位
AND T0240  ; 后腔体出料机械手夹爪张开位
OR H60.07  ; NG处理完成
ANDLD
LDNOT W38.02  ; 到后取料位置
ORNOT W38.01  ; 到前取料位置
ANDLD
ORLD
AND 1491.03  ; 出料伺服到待机位条件
AND 100.02  ; 自动启动
ANDNOT H100.02  ; 错误模拟
AND 1243.11  ; 出料伺服自动定位条件
OUT TR0
AND T0701  ; 出料伺服延时启动
OUT W38.15  ; 伺服运动
LD TR0
TIMX(550) 0701 #1  ; 出料伺服延时启动
; rung 17: NG料处理条件
LD T0000  ; PLC上电
OUT TR0
AND H61.00  ; 1#测试NG有料
AND H60.09  ; 2#测试NG有料
AND H60.14  ; 3#测试NG有料
AND H60.15  ; 4#测试NG有料
NOT(520)
AND W492.01  ; NG传感器信号有空位
OUT W492.00  ; NG位未满
LD TR0
ANDNOT T0148  ; #1测试NG缓存放料位无料感应
ANDNOT T0149  ; #2测试NG缓存放料位无料感应
ANDNOT T0151  ; #4测试NG缓存储料位无料感应延时
ANDNOT T0150  ; #3测试NG缓存储料位无料感应延时
NOT(520)
OUT W492.01  ; NG传感器信号有空位
LD TR0
AND 1497.04  ; 出料到OK/NG位(步)
LD 1490.02  ; 出料伺服在前取料位置
OR 1490.03  ; 出料伺服在后取料位置
OR 1490.01  ; 出料伺服在#1NG位置
ANDLD
AND H60.05  ; NG料在托盘
SET W38.14  ; 有NG 料处理

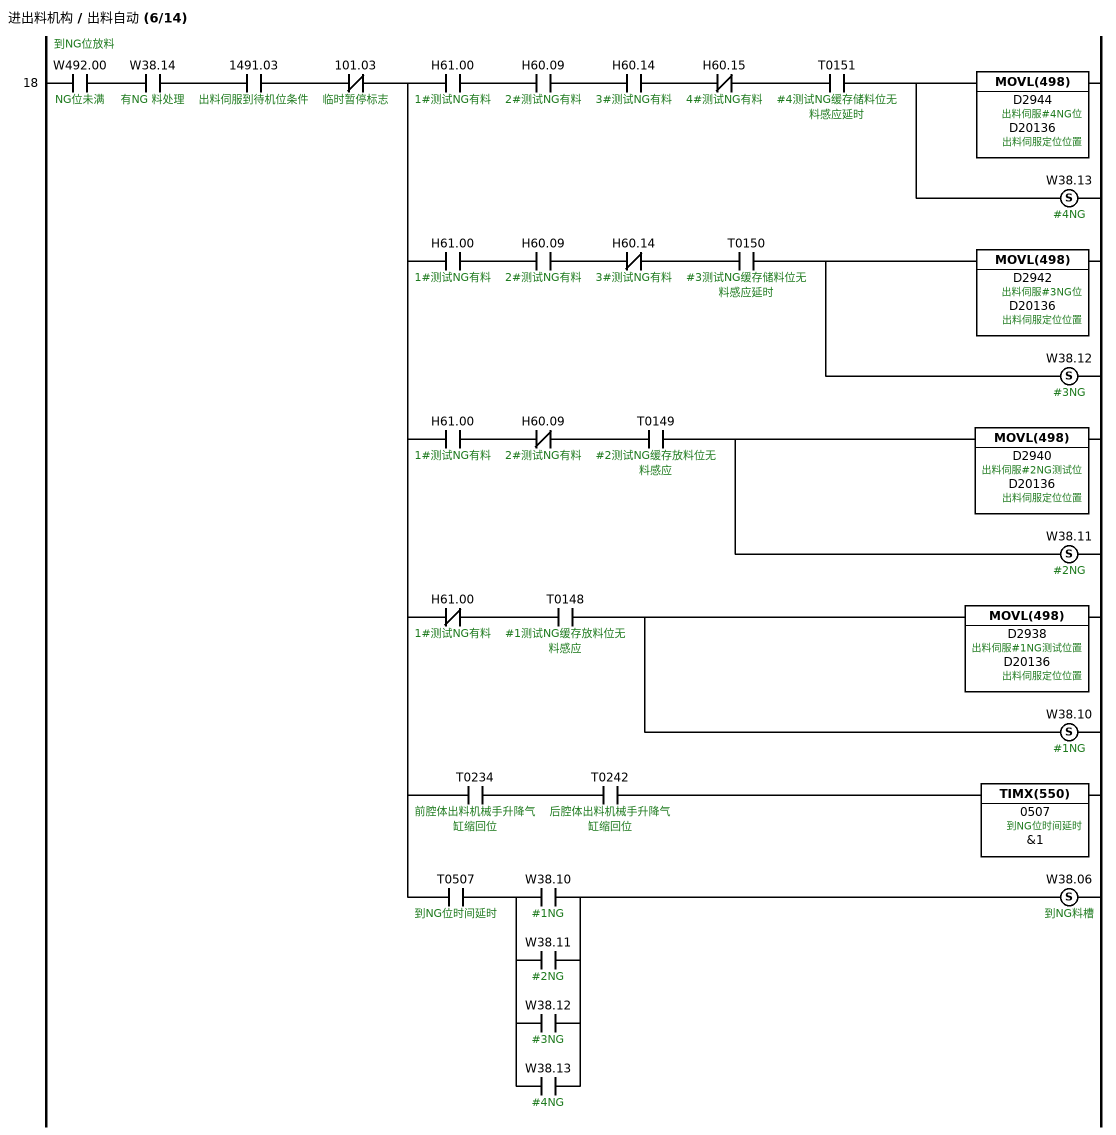
; rung 18: 到NG位放料
LD W492.00  ; NG位未满
AND W38.14  ; 有NG 料处理
AND 1491.03  ; 出料伺服到待机位条件
ANDNOT 101.03  ; 临时暂停标志
OUT TR0
AND H61.00  ; 1#测试NG有料
AND H60.09  ; 2#测试NG有料
AND H60.14  ; 3#测试NG有料
ANDNOT H60.15  ; 4#测试NG有料
AND T0151  ; #4测试NG缓存储料位无料感应延时
MOVL(498) D2944 D20136  ; 出料伺服#4NG位, 出料伺服定位位置
SET W38.13  ; #4NG
LD TR0
AND H61.00  ; 1#测试NG有料
AND H60.09  ; 2#测试NG有料
ANDNOT H60.14  ; 3#测试NG有料
AND T0150  ; #3测试NG缓存储料位无料感应延时
MOVL(498) D2942 D20136  ; 出料伺服#3NG位, 出料伺服定位位置
SET W38.12  ; #3NG
LD TR0
AND H61.00  ; 1#测试NG有料
ANDNOT H60.09  ; 2#测试NG有料
AND T0149  ; #2测试NG缓存放料位无料感应
MOVL(498) D2940 D20136  ; 出料伺服#2NG测试位, 出料伺服定位位置
SET W38.11  ; #2NG
LD TR0
ANDNOT H61.00  ; 1#测试NG有料
AND T0148  ; #1测试NG缓存放料位无料感应
MOVL(498) D2938 D20136  ; 出料伺服#1NG测试位置, 出料伺服定位位置
SET W38.10  ; #1NG
LD TR0
AND T0234  ; 前腔体出料机械手升降气缸缩回位
AND T0242  ; 后腔体出料机械手升降气缸缩回位
TIMX(550) 0507 &1  ; 到NG位时间延时
LD TR0
AND T0507  ; 到NG位时间延时
LD W38.10  ; #1NG
OR W38.11  ; #2NG
OR W38.12  ; #3NG
OR W38.13  ; #4NG
ANDLD
SET W38.06  ; 到NG料槽

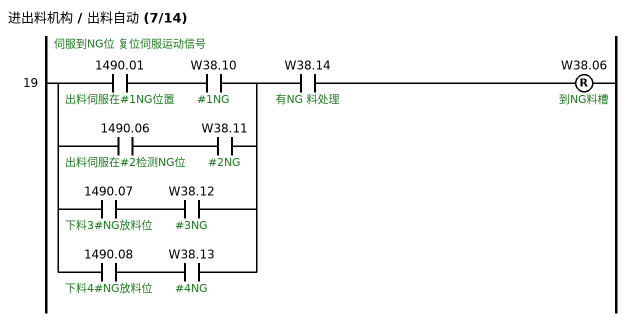
; rung 19: 伺服到NG位 复位伺服运动信号
LD 1490.01  ; 出料伺服在#1NG位置
AND W38.10  ; #1NG
LD 1490.06  ; 出料伺服在#2检测NG位
AND W38.11  ; #2NG
ORLD
LD 1490.07  ; 下料3#NG放料位
AND W38.12  ; #3NG
ORLD
LD 1490.08  ; 下料4#NG放料位
AND W38.13  ; #4NG
ORLD
AND W38.14  ; 有NG 料处理
RSET W38.06  ; 到NG料槽

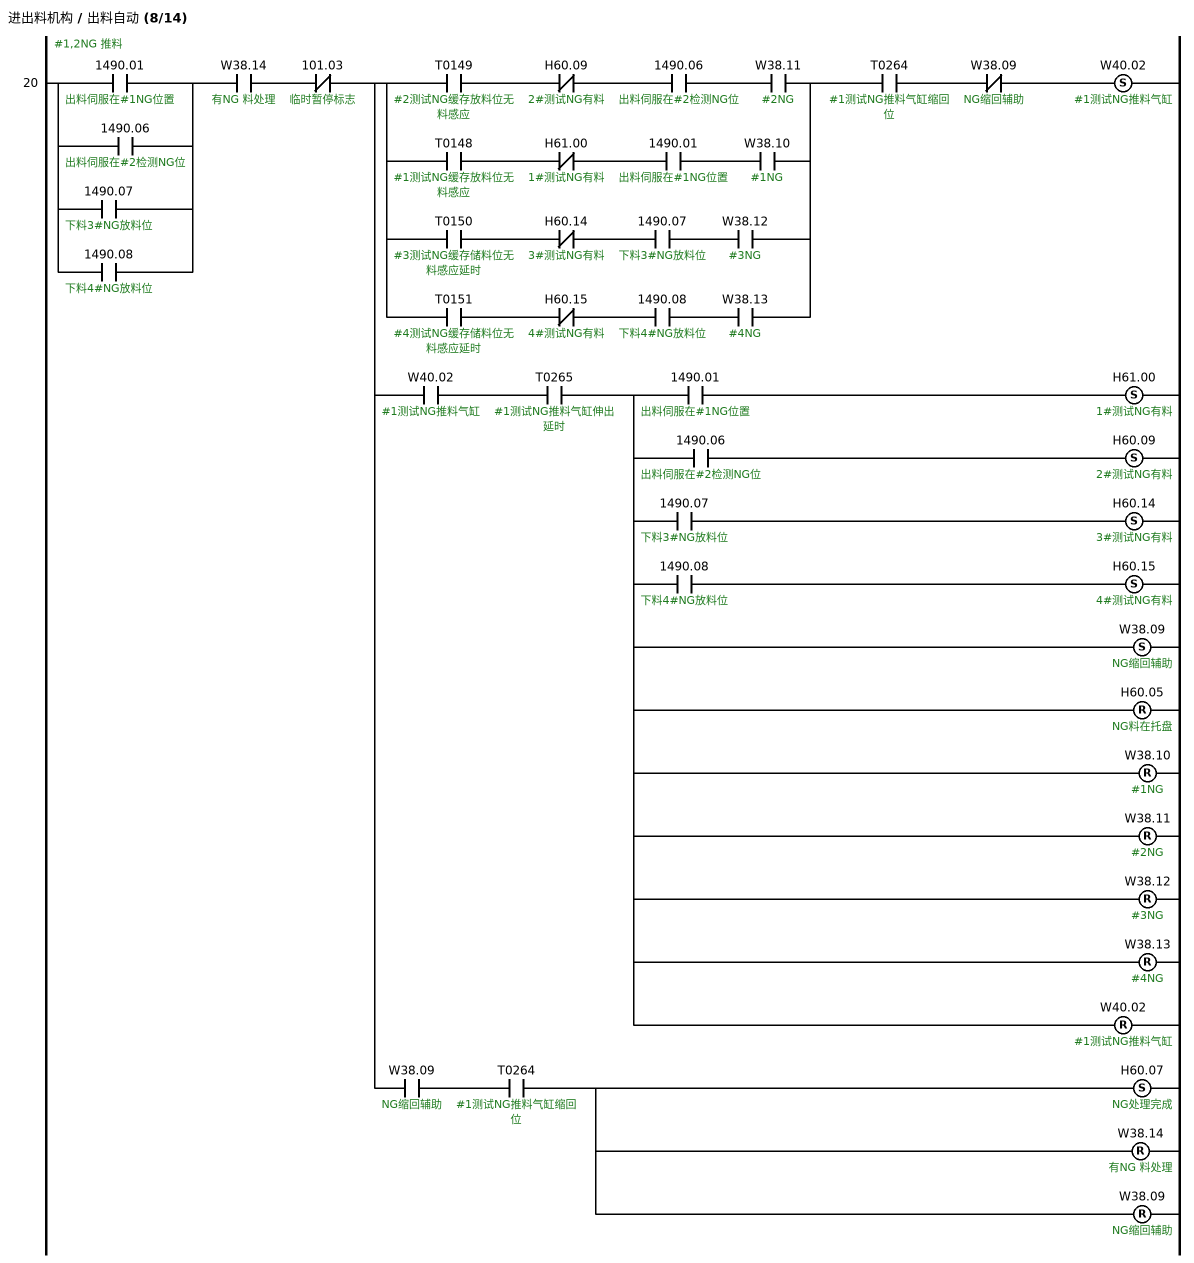
; rung 20: #1,2NG 推料
LD 1490.01  ; 出料伺服在#1NG位置
OR 1490.06  ; 出料伺服在#2检测NG位
OR 1490.07  ; 下料3#NG放料位
OR 1490.08  ; 下料4#NG放料位
AND W38.14  ; 有NG 料处理
ANDNOT 101.03  ; 临时暂停标志
OUT TR0
LD T0149  ; #2测试NG缓存放料位无料感应
ANDNOT H60.09  ; 2#测试NG有料
AND 1490.06  ; 出料伺服在#2检测NG位
AND W38.11  ; #2NG
LD T0148  ; #1测试NG缓存放料位无料感应
ANDNOT H61.00  ; 1#测试NG有料
AND 1490.01  ; 出料伺服在#1NG位置
AND W38.10  ; #1NG
ORLD
LD T0150  ; #3测试NG缓存储料位无料感应延时
ANDNOT H60.14  ; 3#测试NG有料
AND 1490.07  ; 下料3#NG放料位
AND W38.12  ; #3NG
ORLD
LD T0151  ; #4测试NG缓存储料位无料感应延时
ANDNOT H60.15  ; 4#测试NG有料
AND 1490.08  ; 下料4#NG放料位
AND W38.13  ; #4NG
ORLD
ANDLD
AND T0264  ; #1测试NG推料气缸缩回位
ANDNOT W38.09  ; NG缩回辅助
SET W40.02  ; #1测试NG推料气缸
LD TR0
AND W40.02  ; #1测试NG推料气缸
AND T0265  ; #1测试NG推料气缸伸出延时
OUT TR1
AND 1490.01  ; 出料伺服在#1NG位置
SET H61.00  ; 1#测试NG有料
LD TR1
AND 1490.06  ; 出料伺服在#2检测NG位
SET H60.09  ; 2#测试NG有料
LD TR1
AND 1490.07  ; 下料3#NG放料位
SET H60.14  ; 3#测试NG有料
LD TR1
AND 1490.08  ; 下料4#NG放料位
SET H60.15  ; 4#测试NG有料
LD TR1
SET W38.09  ; NG缩回辅助
RSET H60.05  ; NG料在托盘
RSET W38.10  ; #1NG
RSET W38.11  ; #2NG
RSET W38.12  ; #3NG
RSET W38.13  ; #4NG
RSET W40.02  ; #1测试NG推料气缸
LD TR0
AND W38.09  ; NG缩回辅助
AND T0264  ; #1测试NG推料气缸缩回位
SET H60.07  ; NG处理完成
RSET W38.14  ; 有NG 料处理
RSET W38.09  ; NG缩回辅助

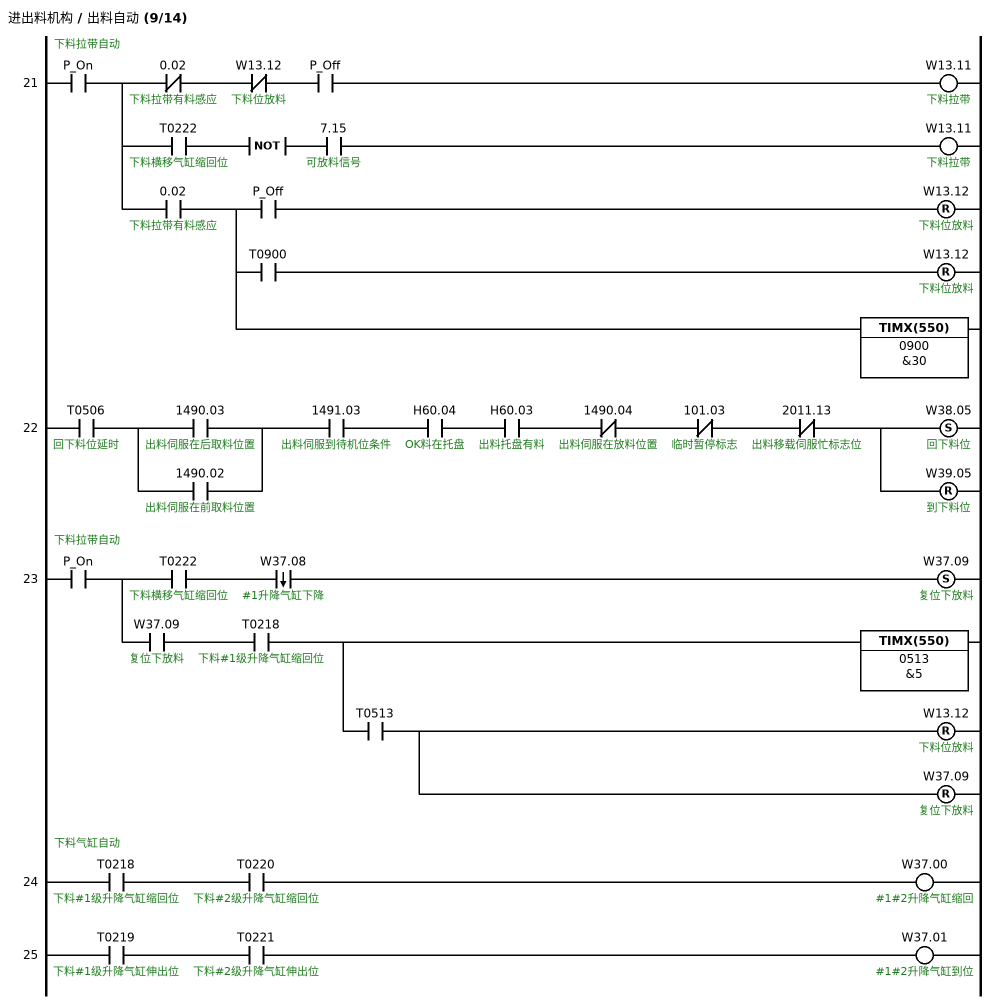
; rung 21: 下料拉带自动
LD P_On
OUT TR0
ANDNOT 0.02  ; 下料拉带有料感应
ANDNOT W13.12  ; 下料位放料
AND P_Off
OUT W13.11  ; 下料拉带
LD TR0
AND T0222  ; 下料横移气缸缩回位
NOT(520)
AND 7.15  ; 可放料信号
OUT W13.11  ; 下料拉带
LD TR0
AND 0.02  ; 下料拉带有料感应
OUT TR0
AND P_Off
RSET W13.12  ; 下料位放料
LD TR0
AND T0900
RSET W13.12  ; 下料位放料
LD TR0
TIMX(550) 0900 &30
; rung 22
LD T0506  ; 回下料位延时
LD 1490.03  ; 出料伺服在后取料位置
OR 1490.02  ; 出料伺服在前取料位置
ANDLD
AND 1491.03  ; 出料伺服到待机位条件
AND H60.04  ; OK料在托盘
AND H60.03  ; 出料托盘有料
ANDNOT 1490.04  ; 出料伺服在放料位置
ANDNOT 101.03  ; 临时暂停标志
ANDNOT 2011.13  ; 出料移载伺服忙标志位
SET W38.05  ; 回下料位
RSET W39.05  ; 到下料位
; rung 23: 下料拉带自动
LD P_On
OUT TR0
AND T0222  ; 下料横移气缸缩回位
%AND W37.08  ; #1升降气缸下降
SET W37.09  ; 复位下放料
LD TR0
AND W37.09  ; 复位下放料
AND T0218  ; 下料#1级升降气缸缩回位
TIMX(550) 0513 &5
AND T0513
RSET W13.12  ; 下料位放料
RSET W37.09  ; 复位下放料
; rung 24: 下料气缸自动
LD T0218  ; 下料#1级升降气缸缩回位
AND T0220  ; 下料#2级升降气缸缩回位
OUT W37.00  ; #1#2升降气缸缩回
; rung 25
LD T0219  ; 下料#1级升降气缸伸出位
AND T0221  ; 下料#2级升降气缸伸出位
OUT W37.01  ; #1#2升降气缸到位

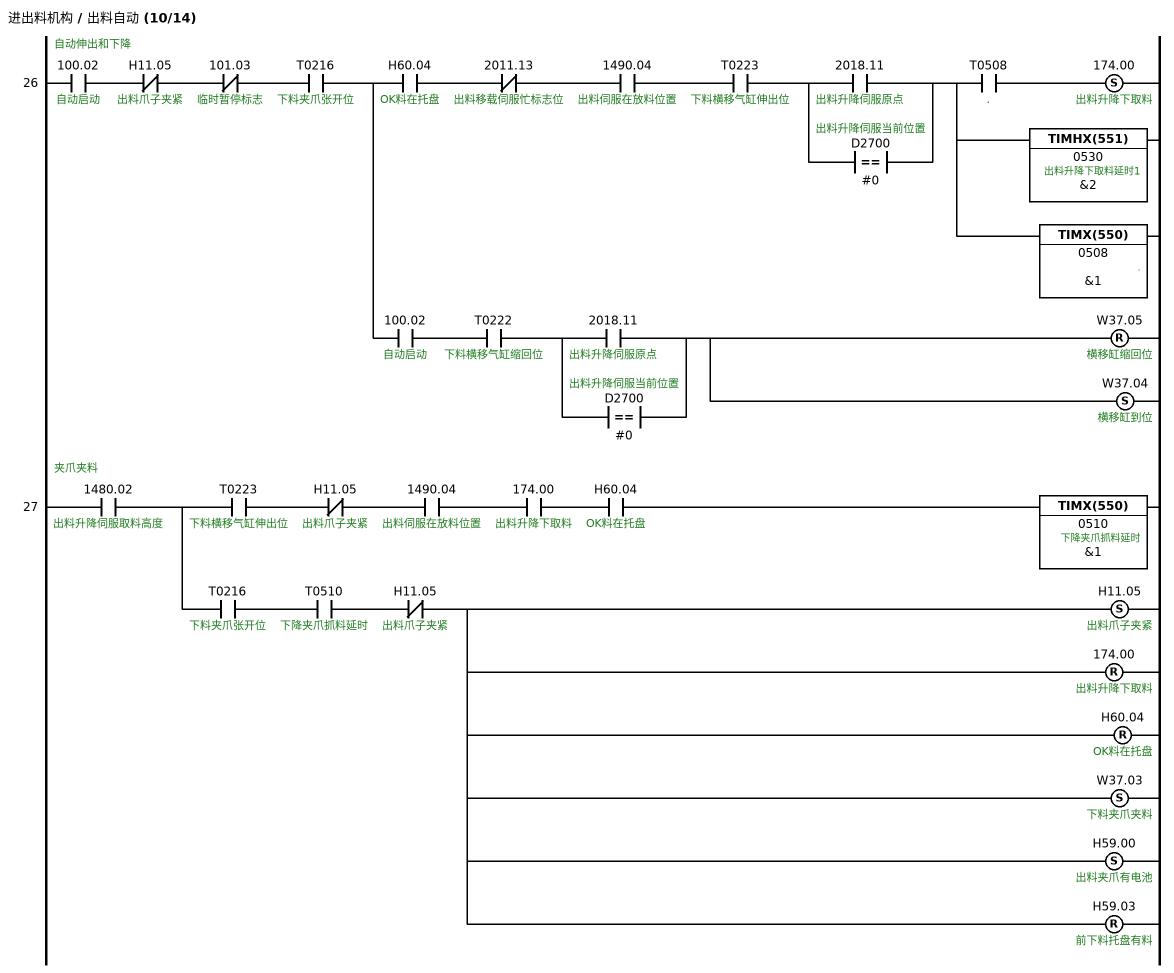
; rung 26: 自动伸出和下降
LD 100.02  ; 自动启动
ANDNOT H11.05  ; 出料爪子夹紧
ANDNOT 101.03  ; 临时暂停标志
AND T0216  ; 下料夹爪张开位
OUT TR0
AND H60.04  ; OK料在托盘
ANDNOT 2011.13  ; 出料移载伺服忙标志位
AND 1490.04  ; 出料伺服在放料位置
AND T0223  ; 下料横移气缸伸出位
LD 2018.11  ; 出料升降伺服原点
OR=L(301) D2700 #0  ; 出料升降伺服当前位置
ANDLD
OUT TR1
AND T0508  ; .
SET 174.00  ; 出料升降下取料
LD TR1
TIMHX(551) 0530 &2  ; 出料升降下取料延时1
TIMX(550) 0508 &1  ; .
LD TR0
AND 100.02  ; 自动启动
AND T0222  ; 下料横移气缸缩回位
LD 2018.11  ; 出料升降伺服原点
OR=L(301) D2700 #0  ; 出料升降伺服当前位置
ANDLD
RSET W37.05  ; 横移缸缩回位
SET W37.04  ; 横移缸到位
; rung 27: 夹爪夹料
LD 1480.02  ; 出料升降伺服取料高度
OUT TR0
AND T0223  ; 下料横移气缸伸出位
ANDNOT H11.05  ; 出料爪子夹紧
AND 1490.04  ; 出料伺服在放料位置
AND 174.00  ; 出料升降下取料
AND H60.04  ; OK料在托盘
TIMX(550) 0510 &1  ; 下降夹爪抓料延时
LD TR0
AND T0216  ; 下料夹爪张开位
AND T0510  ; 下降夹爪抓料延时
ANDNOT H11.05  ; 出料爪子夹紧
SET H11.05  ; 出料爪子夹紧
RSET 174.00  ; 出料升降下取料
RSET H60.04  ; OK料在托盘
SET W37.03  ; 下料夹爪夹料
SET H59.00  ; 出料夹爪有电池
RSET H59.03  ; 前下料托盘有料

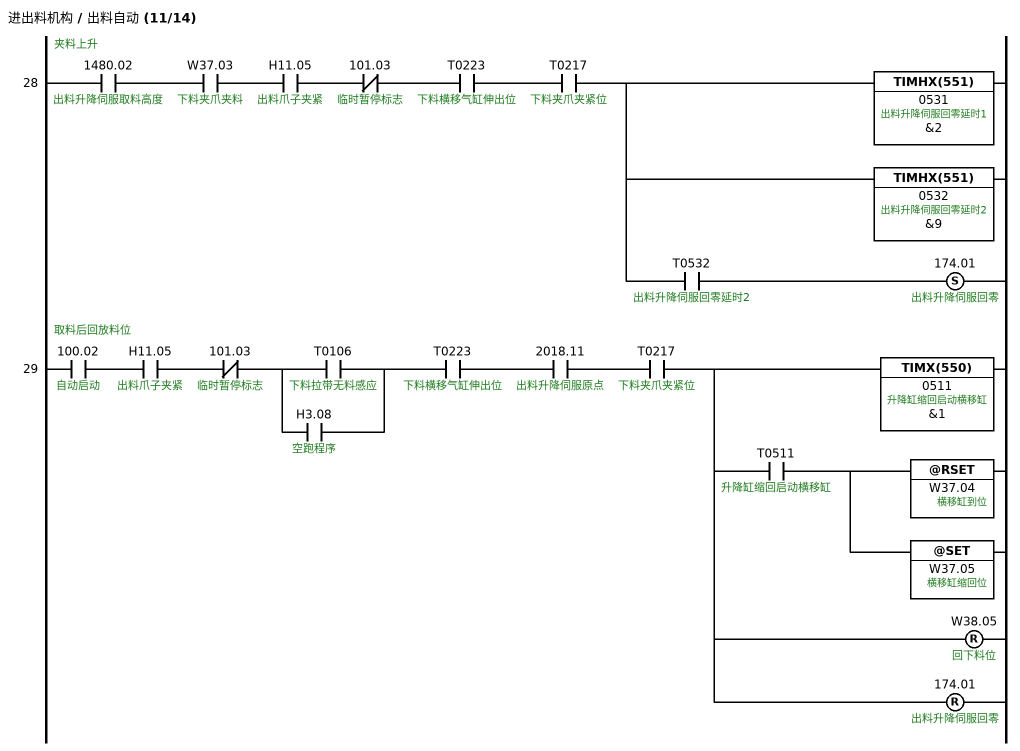
; rung 28: 夹料上升
LD 1480.02  ; 出料升降伺服取料高度
AND W37.03  ; 下料夹爪夹料
AND H11.05  ; 出料爪子夹紧
ANDNOT 101.03  ; 临时暂停标志
AND T0223  ; 下料横移气缸伸出位
AND T0217  ; 下料夹爪夹紧位
TIMHX(551) 0531 &2  ; 出料升降伺服回零延时1
TIMHX(551) 0532 &9  ; 出料升降伺服回零延时2
AND T0532  ; 出料升降伺服回零延时2
SET 174.01  ; 出料升降伺服回零
; rung 29: 取料后回放料位
LD 100.02  ; 自动启动
AND H11.05  ; 出料爪子夹紧
ANDNOT 101.03  ; 临时暂停标志
LD T0106  ; 下料拉带无料感应
OR H3.08  ; 空跑程序
ANDLD
AND T0223  ; 下料横移气缸伸出位
AND 2018.11  ; 出料升降伺服原点
AND T0217  ; 下料夹爪夹紧位
OUT TR0
TIMX(550) 0511 &1  ; 升降缸缩回启动横移缸
AND T0511  ; 升降缸缩回启动横移缸
@RSET W37.04  ; 横移缸到位
@SET W37.05  ; 横移缸缩回位
LD TR0
RSET W38.05  ; 回下料位
RSET 174.01  ; 出料升降伺服回零

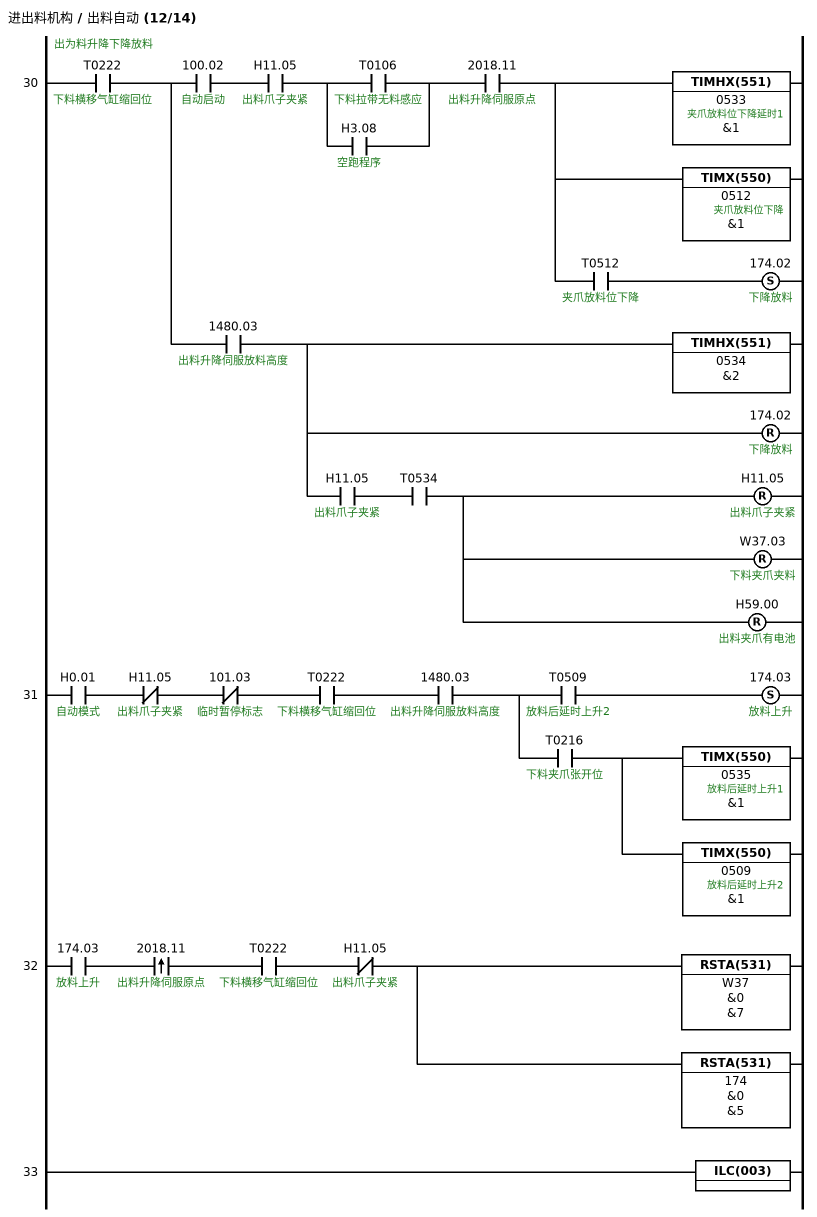
; rung 30: 出为料升降下降放料
LD T0222  ; 下料横移气缸缩回位
OUT TR0
AND 100.02  ; 自动启动
AND H11.05  ; 出料爪子夹紧
LD T0106  ; 下料拉带无料感应
OR H3.08  ; 空跑程序
ANDLD
AND 2018.11  ; 出料升降伺服原点
TIMHX(551) 0533 &1  ; 夹爪放料位下降延时1
TIMX(550) 0512 &1  ; 夹爪放料位下降
AND T0512  ; 夹爪放料位下降
SET 174.02  ; 下降放料
LD TR0
AND 1480.03  ; 出料升降伺服放料高度
TIMHX(551) 0534 &2
RSET 174.02  ; 下降放料
AND H11.05  ; 出料爪子夹紧
AND T0534
RSET H11.05  ; 出料爪子夹紧
RSET W37.03  ; 下料夹爪夹料
RSET H59.00  ; 出料夹爪有电池
; rung 31
LD H0.01  ; 自动模式
ANDNOT H11.05  ; 出料爪子夹紧
ANDNOT 101.03  ; 临时暂停标志
AND T0222  ; 下料横移气缸缩回位
AND 1480.03  ; 出料升降伺服放料高度
OUT TR0
AND T0509  ; 放料后延时上升2
SET 174.03  ; 放料上升
LD TR0
AND T0216  ; 下料夹爪张开位
TIMX(550) 0535 &1  ; 放料后延时上升1
TIMX(550) 0509 &1  ; 放料后延时上升2
; rung 32
LD 174.03  ; 放料上升
@AND 2018.11  ; 出料升降伺服原点
AND T0222  ; 下料横移气缸缩回位
ANDNOT H11.05  ; 出料爪子夹紧
RSTA(531) W37 &0 &7
RSTA(531) 174 &0 &5
; rung 33
ILC(003)

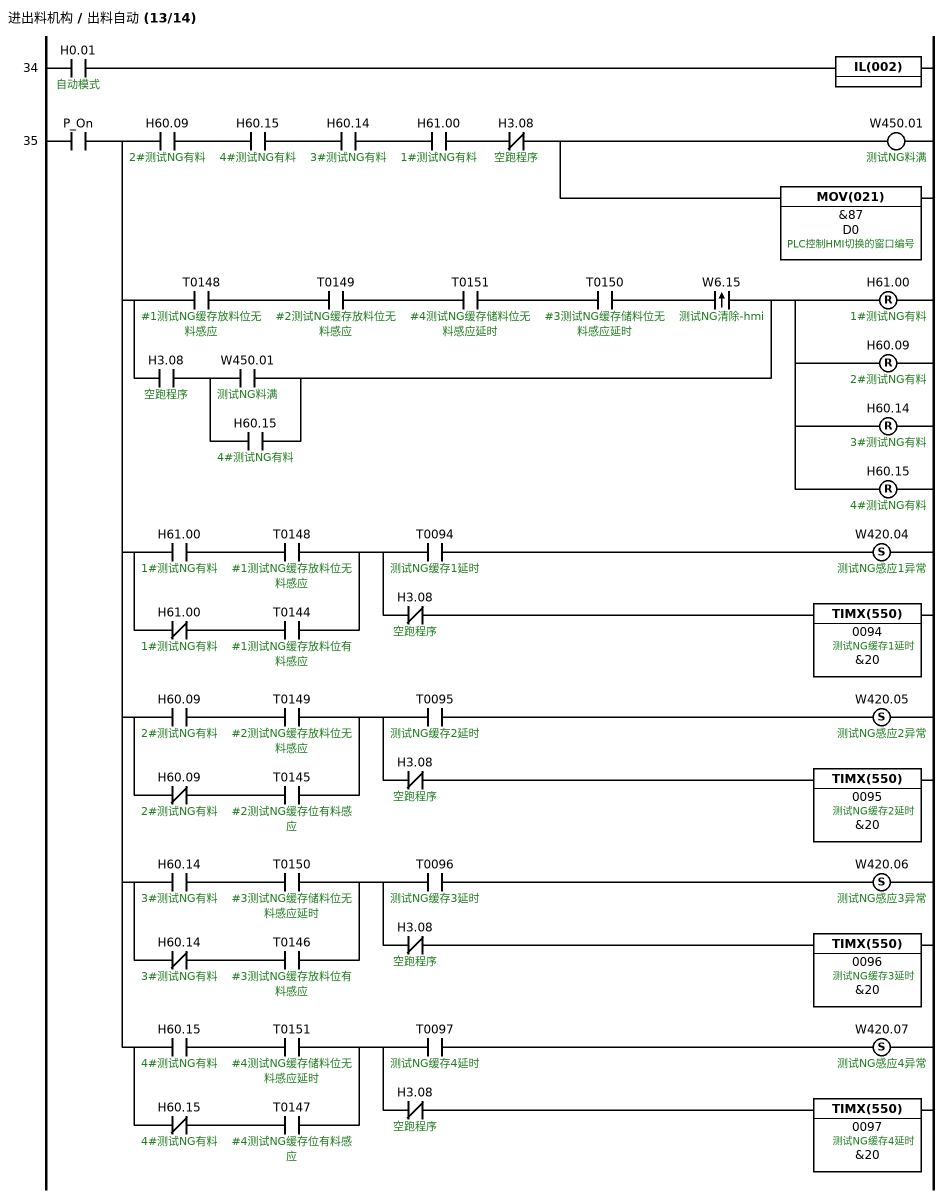
; rung 34
LD H0.01  ; 自动模式
IL(002)
; rung 35
LD P_On
OUT TR0
AND H60.09  ; 2#测试NG有料
AND H60.15  ; 4#测试NG有料
AND H60.14  ; 3#测试NG有料
AND H61.00  ; 1#测试NG有料
ANDNOT H3.08  ; 空跑程序
OUT W450.01  ; 测试NG料满
MOV(021) &87 D0  ; PLC控制HMI切换的窗口编号
LD TR0
LD T0148  ; #1测试NG缓存放料位无料感应
AND T0149  ; #2测试NG缓存放料位无料感应
AND T0151  ; #4测试NG缓存储料位无料感应延时
AND T0150  ; #3测试NG缓存储料位无料感应延时
@AND W6.15  ; 测试NG清除-hmi
LD H3.08  ; 空跑程序
LD W450.01  ; 测试NG料满
OR H60.15  ; 4#测试NG有料
ANDLD
ORLD
ANDLD
RSET H61.00  ; 1#测试NG有料
RSET H60.09  ; 2#测试NG有料
RSET H60.14  ; 3#测试NG有料
RSET H60.15  ; 4#测试NG有料
LD TR0
LD H61.00  ; 1#测试NG有料
AND T0148  ; #1测试NG缓存放料位无料感应
LDNOT H61.00  ; 1#测试NG有料
AND T0144  ; #1测试NG缓存放料位有料感应
ORLD
ANDLD
OUT TR1
AND T0094  ; 测试NG缓存1延时
SET W420.04  ; 测试NG感应1异常
LD TR1
ANDNOT H3.08  ; 空跑程序
TIMX(550) 0094 &20  ; 测试NG缓存1延时
LD TR0
LD H60.09  ; 2#测试NG有料
AND T0149  ; #2测试NG缓存放料位无料感应
LDNOT H60.09  ; 2#测试NG有料
AND T0145  ; #2测试NG缓存位有料感应
ORLD
ANDLD
OUT TR1
AND T0095  ; 测试NG缓存2延时
SET W420.05  ; 测试NG感应2异常
LD TR1
ANDNOT H3.08  ; 空跑程序
TIMX(550) 0095 &20  ; 测试NG缓存2延时
LD TR0
LD H60.14  ; 3#测试NG有料
AND T0150  ; #3测试NG缓存储料位无料感应延时
LDNOT H60.14  ; 3#测试NG有料
AND T0146  ; #3测试NG缓存放料位有料感应
ORLD
ANDLD
OUT TR1
AND T0096  ; 测试NG缓存3延时
SET W420.06  ; 测试NG感应3异常
LD TR1
ANDNOT H3.08  ; 空跑程序
TIMX(550) 0096 &20  ; 测试NG缓存3延时
LD TR0
LD H60.15  ; 4#测试NG有料
AND T0151  ; #4测试NG缓存储料位无料感应延时
LDNOT H60.15  ; 4#测试NG有料
AND T0147  ; #4测试NG缓存位有料感应
ORLD
ANDLD
OUT TR0
AND T0097  ; 测试NG缓存4延时
SET W420.07  ; 测试NG感应4异常
LD TR0
ANDNOT H3.08  ; 空跑程序
TIMX(550) 0097 &20  ; 测试NG缓存4延时

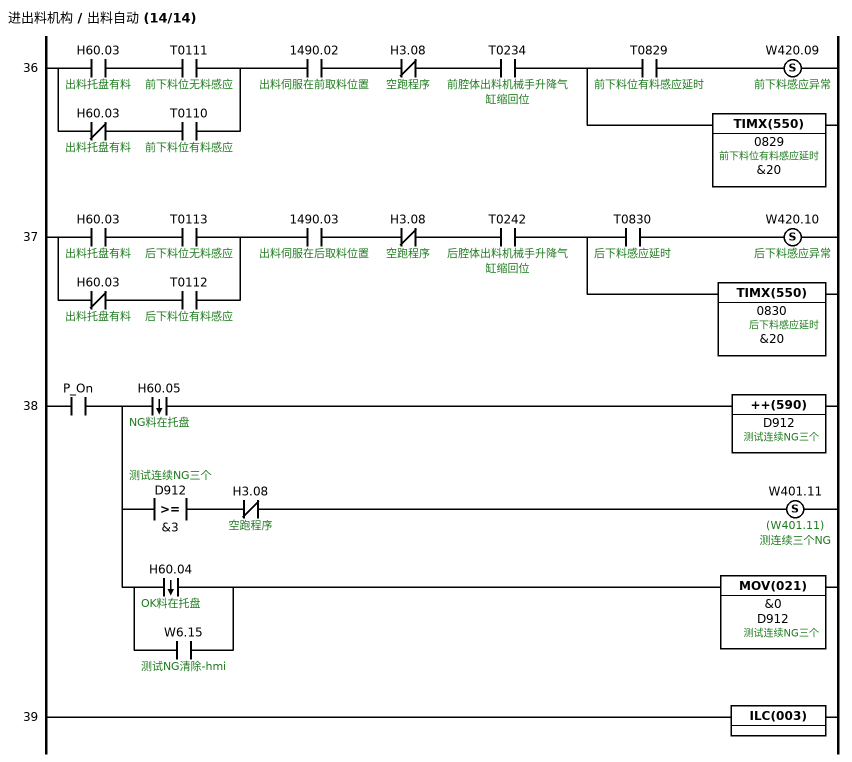
; rung 36
LD H60.03  ; 出料托盘有料
AND T0111  ; 前下料位无料感应
LDNOT H60.03  ; 出料托盘有料
AND T0110  ; 前下料位有料感应
ORLD
AND 1490.02  ; 出料伺服在前取料位置
ANDNOT H3.08  ; 空跑程序
AND T0234  ; 前腔体出料机械手升降气缸缩回位
OUT TR0
AND T0829  ; 前下料位有料感应延时
SET W420.09  ; 前下料感应异常
LD TR0
TIMX(550) 0829 &20  ; 前下料位有料感应延时
; rung 37
LD H60.03  ; 出料托盘有料
AND T0113  ; 后下料位无料感应
LDNOT H60.03  ; 出料托盘有料
AND T0112  ; 后下料位有料感应
ORLD
AND 1490.03  ; 出料伺服在后取料位置
ANDNOT H3.08  ; 空跑程序
AND T0242  ; 后腔体出料机械手升降气缸缩回位
OUT TR0
AND T0830  ; 后下料感应延时
SET W420.10  ; 后下料感应异常
LD TR0
TIMX(550) 0830 &20  ; 后下料感应延时
; rung 38
LD P_On
OUT TR0
%AND H60.05  ; NG料在托盘
++(590) D912  ; 测试连续NG三个
LD TR0
AND>=(325) D912 &3  ; 测试连续NG三个
ANDNOT H3.08  ; 空跑程序
SET W401.11  ; (W401.11) 测连续三个NG
LD TR0
%LD H60.04  ; OK料在托盘
OR W6.15  ; 测试NG清除-hmi
ANDLD
MOV(021) &0 D912  ; 测试连续NG三个
; rung 39
ILC(003)

### Section 外部输出

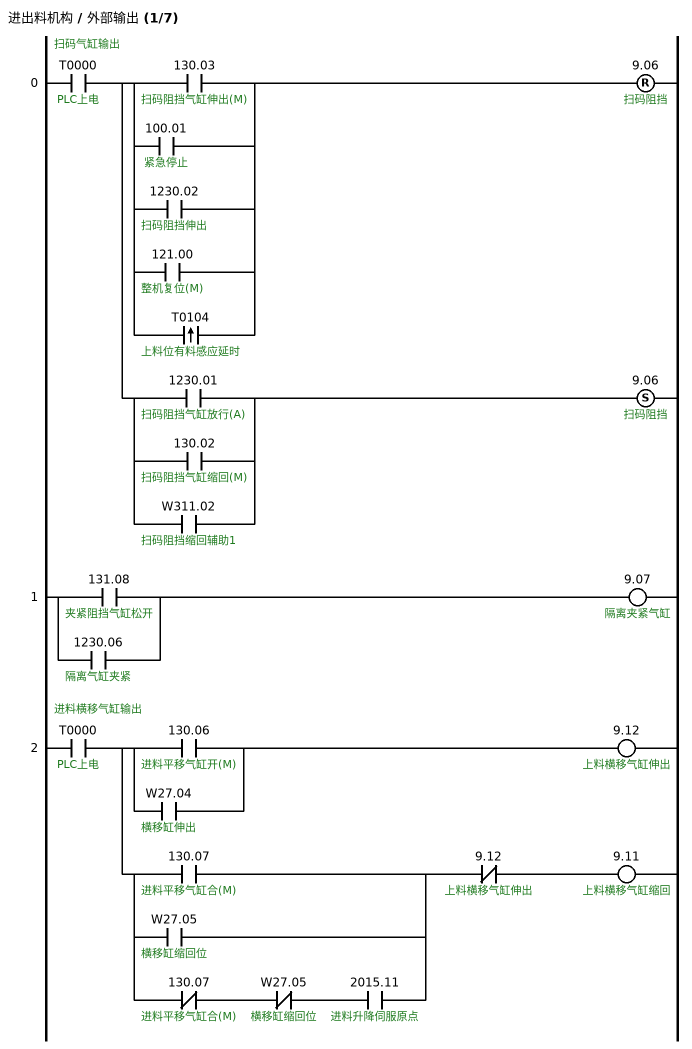
; rung 0: 扫码气缸输出
LD T0000  ; PLC上电
OUT TR0
LD 130.03  ; 扫码阻挡气缸伸出(M)
OR 100.01  ; 紧急停止
OR 1230.02  ; 扫码阻挡伸出
OR 121.00  ; 整机复位(M)
@OR T0104  ; 上料位有料感应延时
ANDLD
RSET 9.06  ; 扫码阻挡
LD TR0
LD 1230.01  ; 扫码阻挡气缸放行(A)
OR 130.02  ; 扫码阻挡气缸缩回(M)
OR W311.02  ; 扫码阻挡缩回辅助1
ANDLD
SET 9.06  ; 扫码阻挡
; rung 1
LD 131.08  ; 夹紧阻挡气缸松开
OR 1230.06  ; 隔离气缸夹紧
OUT 9.07  ; 隔离夹紧气缸
; rung 2: 进料横移气缸输出
LD T0000  ; PLC上电
OUT TR0
LD 130.06  ; 进料平移气缸开(M)
OR W27.04  ; 横移缸伸出
ANDLD
OUT 9.12  ; 上料横移气缸伸出
LD TR0
LD 130.07  ; 进料平移气缸合(M)
OR W27.05  ; 横移缸缩回位
LDNOT 130.07  ; 进料平移气缸合(M)
ANDNOT W27.05  ; 横移缸缩回位
AND 2015.11  ; 进料升降伺服原点
ORLD
ANDLD
ANDNOT 9.12  ; 上料横移气缸伸出
OUT 9.11  ; 上料横移气缸缩回

